           //#sendBuffer.Header.SessionHandle := DWORD_TO_DINT(SWAP(DINT_TO_DWORD(#Config.currentSessionID)));
           #sendBuffer.Header.SessionHandle := DWORD_TO_DINT( SHL(IN := DINT_TO_DWORD(#Config.currentSessionID), N := 24) OR
                                                             (SHL(IN := DINT_TO_DWORD(#Config.currentSessionID), N :=  8) AND DW#16#00FF0000) OR
                                                             (SHR(IN := DINT_TO_DWORD(#Config.currentSessionID), N :=  8) AND DW#16#0000FF00) OR
                                                              SHR(IN := DINT_TO_DWORD(#Config.currentSessionID), N := 24));
           #sendBuffer.Header.Status := 0;
           #sendBuffer.Header.Options := 0;
           //the Context will be a combination out of the own instance identifier
           //and a sequence number
           #sendBuffer.Header.Context[1] := DWORD_TO_BYTE(DINT_TO_DWORD(#ownInstance) AND DW#16#000000FF);
           #sendBuffer.Header.Context[2] := DWORD_TO_BYTE(SHR(IN := DINT_TO_DWORD(#ownInstance), N := 8) AND DW#16#000000FF);
           #sendBuffer.Header.Context[3] := DWORD_TO_BYTE(SHR(IN := DINT_TO_DWORD(#ownInstance), N := 16) AND DW#16#000000FF);
           #sendBuffer.Header.Context[4] := DWORD_TO_BYTE(SHR(IN := DINT_TO_DWORD(#ownInstance), N := 24) AND DW#16#000000FF);
           #sendBuffer.Header.Context[5] := DWORD_TO_BYTE(DINT_TO_DWORD(#ownSequence) AND DW#16#000000FF);
           #sendBuffer.Header.Context[6] := DWORD_TO_BYTE(SHR(IN := DINT_TO_DWORD(#ownSequence), N := 8) AND DW#16#000000FF);
           #sendBuffer.Header.Context[7] := DWORD_TO_BYTE(SHR(IN := DINT_TO_DWORD(#ownSequence), N := 16) AND DW#16#000000FF);
           #sendBuffer.Header.Context[8] := DWORD_TO_BYTE(SHR(IN := DINT_TO_DWORD(#ownSequence), N := 24) AND DW#16#000000FF);
           #sendBuffer.Data[1] := 16#00;

           //Checking the MuteEx
           IF #Config.instanceLock = 0 OR
             #Config.instanceLock = #ownInstance
           THEN
             //Locking the MutEx
             #Config.instanceLock := #ownInstance;
             #send.LEN := #EIP_HEADER_LENGTH;
             #send.REQ := TRUE;
             // Action
             // 

             #send(ID := #connection.id,
                   DATA := #sendBuffer);

             // Transition
             //
             #internalState := #STATE_UNREGISTERING;
             #Config.references := #Config.references - 1;
           ELSE
             IF #Config.instanceLock = #ownInstance THEN
               #Config.instanceLock := 0;
             END_IF;
           END_IF;

         ELSE
           IF #Config.references > 1 THEN
             #Config.references := #Config.references - 1;
           END_IF;
           #internalState := #STATE_POWER_OFF;
         END_IF;

       #STATE_UNREGISTERING:
         // Action
         // 

         #send(ID := #connection.id,
               DATA := #sendBuffer);

         // Transition
         //
         IF #send.STATUS = #RESULT_JOB_START THEN
           ;
         ELSIF #send.STATUS = #RESULT_JOB_RUNNING THEN
           #send.REQ := FALSE;

         ELSIF #send.STATUS = #RESULT_SUCCESS THEN
           #send.REQ := FALSE;
           #internalState := #STATE_DISCONNECTING;
           //Unlocking MuteEx
           #Config.instanceLock := 0;
         ELSE

           #Status := W#16#8200 OR (#send.STATUS AND 16#00FF);
           #send.REQ := FALSE;
           #internalState := #STATE_DISCONNECTING;
         END_IF;

       #STATE_DISCONNECTING:
         IF #disconnect.STATUS = #RESULT_JOB_START THEN
           #connectionStatus.isConnected := FALSE;
           #connectionStatus.isDisconnecting := TRUE;

         ELSIF #disconnect.STATUS = #RESULT_IDLE THEN
           #connectionStatus.isDisconnecting := TRUE;
           #disconnect.REQ := NOT #disconnect.REQ;

         ELSIF #disconnect.STATUS = #RESULT_JOB_RUNNING THEN
           #disconnect.REQ := FALSE;

         ELSIF #disconnect.STATUS = #RESULT_JOB_NOT_REQUIRED OR
           #disconnect.STATUS = #RESULT_SUCCESS
         THEN
           #disconnect.REQ := FALSE;
           #connectionStatus.isConnected := FALSE;
           #connectionStatus.isDisconnecting := FALSE;
           #connectionStatus.isDisconnected := TRUE;
           #connectionStatus.hasReceivedData := FALSE;
           #connectionStatus.hasReceivedHeader := FALSE;

           #ownInstance := 0;
           #ownSequence := 0;
           #Config.connID := 0;

           #internalState := #STATE_IDLE;
         ELSE
           // Throw error !
           //   Error from disconnecting
           #Status := W#16#8400 OR (#disconnect.STATUS AND 16#00FF);
           #disconnect.REQ := FALSE;
           #connectionStatus.isConnected := FALSE;
           #connectionStatus.isDisconnecting := FALSE;
           #connectionStatus.isDisconnected := TRUE;
           #connectionStatus.hasReceivedData := FALSE;
           #connectionStatus.hasReceivedHeader := FALSE;

           #ownInstance := 0;
           #ownSequence := 0;

           #internalState := #STATE_IDLE;
         END_IF;
       ELSE
         // Throw error !
         //   unknown internal state        
         #Status := W#16#8C00 OR (INT_TO_WORD(#internalState) AND W#16#00FF);
     END_CASE;
   END_IF;

   #previousRequest := #REQ;
   #EnabledJ := #Enable;
END_FUNCTION_BLOCK

// folder: GET_PUT_R

FUNCTION_BLOCK "PUT_R"   // FB6, SCL
{ S7_Optimized_Access := 'TRUE' }
VERSION : 1.0
   VAR_INPUT
      Enable : Bool;   // [TRUE| FALSE] TRUE signal keeps the block in PowerOff state
      REQ : Bool;   // [TRUE |FALSE] rising edge triggers a read request
      InterfaceId : Hw_Interface;   // [1..] InterfaceID of the used interface
      IPv4 : IP_V4;   // [IPv4 address] - shall be in the same subnet as controller is
      Slot : Int;   // [-1..16] -1, when directly connected suc has CompactLogix
   END_VAR
   VAR_OUTPUT
      Status : Word;   // [Enum] status information
      Done : Bool;   // [TRUE | FALSE] TRUE signal is a one shot signal indicating the transmission of the data
      Connecting : Bool;   // [TRUE | FALSE] TRUE signal indicates the establishment of the connection
      Established : Bool;   // [TRUE | FALSE] TRUE indicates an established connection
   END_VAR
   VAR_IN_OUT
      Config : "RockwellConfig";
      Tag : "RockwellTag";   // [RockwelTag] datatype containing the tagname, value and data type
      Value : Variant;
   END_VAR
   VAR
      internalState : UInt;   // [Enum] contains the internal state information
      connect : TCON;
      disconnect : TDISCON;
      send : TSEND;
      receive : TRCV;
      diag : T_DIAG;
      connection : TCON_IP_v4;
      sendBuffer : Struct
         Header : Struct
            Command : Word;   // Encapsulation command
            Length : UInt;   // Length, in bytes, of the command specific data portion of the message
            SessionHandle : UDInt;   // Session identification
            Status : UDInt;   // Status code
            Context : Array[1..8] of USInt;   // Information pertinien only to the sender of an encapsulation command
            Options : UDInt;
         END_STRUCT;
         Data : Array[1..508] of USInt;
      END_STRUCT;
      receiveBuffer : Struct
         Header : Struct
            Command : Word;   // Encapsulation command
            Length : UInt;   // Length, in bytes, of the command specific data portion of the message
            SessionHandle : UDInt;   // Session identification
            Status : UDInt;   // Status code
            Context : Array[1..8] of USInt;   // Information pertinien only to the sender of an encapsulation command
            Options : UDInt;
         END_STRUCT;
         Data : Array[1..508] of USInt;
      END_STRUCT;
      currentResponse : Word;
      connectionStatus : Struct
         isDisconnected : Bool;
         isDisconnecting : Bool;
         isConnecting : Bool;
         isConnected : Bool;
         hasReceivedData : Bool;
         hasReceivedHeader : Bool;
      END_STRUCT;
      indexTag : Int := 0;
      currentCIPService : Byte;
      previousRequest : Bool;
      EnabledJ : Bool;
      ownInstance : DInt;
      ownSequence : DInt;
      diagStatus : TDiag_StatusExt;
      randomGenerator : Struct   // [STRUCT] used to realize a pseudo random number
         m_w : DInt;
         m_z : DInt;
         Val : DInt;
         currentTime : DTL;
         currentMilliSeconds : DInt;
      END_STRUCT;
   END_VAR
   VAR_TEMP
      indexTagName : DInt;
      result : Int;
      itemLength : DInt;   // contains the Length of the EIP packet
      overallLength : DInt;   // contains the Length of the EIP packet
      tagNameLength : DInt;   // contains the Length of the Tagname (in WORDS)
      tagValueLength : DInt;   // contains the Length of the Tag Value
      unconnectedDataItemLength : DInt;   // contains the Length of the unconnected data item
      baseIndexOuterCIPMessage : DInt;   // contains the base index to the beginning of the outer CIP message
      baseIndexInnerCIPMessage : DInt;   // contains the base index to the beginning of the inner CIP message
      receivedServiceStatus : Int;
      receivedInstance : DInt;
      receivedSequence : DInt;
      receivedType : Word;
      valueIndex : Int;
      sendValue : Struct
         Boolean : Bool;
         Short : SInt;
         Integer : Int;
         Double : DInt;
         Float : Real;
      END_STRUCT;
   END_VAR
   VAR CONSTANT
      EIP_VENDOR_ID : Word := 1251;   // EtherNet/IP vendor ID 'Siemens AG'
      EIP_HEADER_LENGTH : UInt := 24;   // EtherNet/IP Encapsulation Header length is 24 bytes
      EIP_PORT : Word := 44818;   // EtherNet/IP standard port is 44818 (0xAF12)
      RESULT_SUCCESS : Word := 16#0000;
      RESULT_IDLE : Word := 16#7000;
      RESULT_JOB_START : Word := 16#7001;
      RESULT_JOB_RUNNING : Word := 16#7002;
      RESULT_JOB_NOT_REQUIRED : Word := 16#80A3;
      RESULT_MORE_AVAIL : Word := 16#80B1;
      RESULT_REUSED_ID : Word := 16#8085;
      EIP_STATUS_OK : UDInt := 0;   // EIP Status OK
      EIP_STATUS_TOOMANY_SESSIONS : UDInt := 16#01000000;   // EIP Status "more than 1 active session on the same TCP connection"
      EIP_STATUS_OUTOFRESSOURCES : UDInt := 16#02000000;   // EIP Status "does not have sufficient resources"
      EIP_STATUS_INVALID_SESSION_ID : UDInt := 16#64000000;   // EIP Status "Invalid Session ID"
      EIP_STATUS_PROTOCOL_ERROR : UDInt := 16#69000000;   // EIP Status "Protocol Version or Options mismatches"
      EIP_CMD_REG_SESSION : Word := 16#0065;   // EtherNet/IP Encapsulation Command "Register Session"
      EIP_CMD_UNREG_SESSION : Word := 16#0066;   // EtherNet/IP Encapsulation Command "Unregister Session"
      EIP_CMD_SEND_RR : Word := 16#006F;   // EtherNet/IP Encapsulation Command "Send RR Data"
      CIP_SRV_TABLEREAD : Byte := 16#4C;   // CIP Service Data Table Read
      CIP_SRV_TABLEWRITE : Byte := 16#4D;   // CIP Service Data Table Write
      CIP_SRV_TABLEREAD_FRAG : Byte := 16#52;   // CIP Service Fragmented Data Table Read
      CIP_SRV_TABLEWRITE_FRAG : Byte := 16#53;   // CIP Service Fragmented Data Table Write
      CIP_SRV_UNCONNECTED_SEND : Byte := 16#52;   // CIP Service Unconnected Send Data
      STATE_IDLE : UInt := 1;
      STATE_INIT : UInt := 2;
      STATE_CONNECTING : UInt := 3;
      STATE_DISCONNECTING : UInt := 4;
      STATE_SENDING : UInt := 5;
      STATE_REGISTER_SESSION : UInt := 6;
      STATE_UNREGISTER_SESSION : UInt := 7;
      STATE_REGISTERING : UInt := 8;
      STATE_UNREGISTERING : UInt := 9;
      STATE_REGISTERED : UInt := 10;
      STATE_SEND : UInt := 11;
      STATE_RECEIVE_HEADER : UInt := 12;
      STATE_RECEIVE_DATA : UInt := 13;
      STATE_POWER_OFF : UInt := 0;
      DT_BOOLEAN_ATOMIC : USInt := 16#C1;
      DT_SINT_ATOMIC : USInt := 16#C2;
      DT_INT_ATOMIC : USInt := 16#C3;
      DT_DINT_ATOMIC : USInt := 16#C4;
      DT_FLOAT_ATOMIC : USInt := 16#CA;
      CIP_PATH_SEG_TYPE_CLASS : USInt := 16#20;
      CIP_PATH_SEG_TYPE_INSTANCE : USInt := 16#24;
      CIP_PATH_SEG_TYPE_ANSI : USInt := 16#91;
      CIP_PATH_SEG_TYPE_PORT : USInt := 16#01;
      CIP_ROUTE_SEG_LENGTH : Int := 4;
      CIP_ROUTE_PATH_LENGTH : Int := 1;
      CIP_TABLEREAD_LENGTH : Int := 6;
      CIP_TABLEWRITE_LENGTH : Int := 4;
      CIP_UCSEND_HEADER_LENGTH : Int := 4;
      CIP_UCSEND_SEG_LENGTH : Int := 6;
      EIP_CMD_SEND_RR_SEG_LENGTH : Int := 16;
      CON_TYPE_TCP_V2 : USInt := 17;   // TCP connection for TCON_PARAM descriptor
      CON_TYPE_TCP_V4 : Byte := 11;   // TCP connection for TCON_IP_V4 descriptor
      CIP_GENSTS_SUCCESS : USInt := 16#00;
      CIP_GENSTS_PATH_SEG_ERROR : USInt := 16#04;
      CIP_GENSTS_PATH_DEST_UNKNOWN : USInt := 16#05;
      CIP_GENSTS_PARTIAL : USInt := 16#06;
      CIP_GENSTS_NOT_ENOUGH_DATA : USInt := 16#13;
      CIP_GENSTS_PATH_SIZE_MISMATCH : USInt := 16#26;
      CIP_GENSTS_DOESNT_EXIST : USInt := 16#16;
      CIP_GENSTS_GENERIC : USInt := 16#FF;
      CIP_SRVSTS_RANGE_EXCEED : UInt := 16#2105;
      CIP_SRVSTS_TYPE_MISMATCH : UInt := 16#2107;
   END_VAR
BEGIN
   //=============================================================================
   // Siemens AG
   // (c)Copyright 2016 All Rights Reserved
   //-----------------------------------------------------------------------------
   // Library: PutGet_Rockwell
   // Tested with: 1511-1 PN V1.8.3 and ControlLogix/Compactlogix
   // Engineering: TIA Portal V13 SP1 Upd 9
   // Restrictions: look into pdf
   // Requirements: S7-1500 V1.8.3
   // Functionality: Get Put Values from to Rockwell CPU
   //-----------------------------------------------------------------------------
   // Change log table:
   // Version  Date            Expert in charge        Changes applied
   // 01.00.01 12.07.2016      Scheel                  initial version 
   // 01.00.02 22.07.2016      Scheel                  feat: add diagnostics and
   //                                                        indicators
   // 01.00.03 22.07.2016      Scheel                  fix: diagnostics indicators
   // 01.00.04 19.10.2016      Scheel                  fix: connect will be
   //                                                       retriggered, when idle
   //                                                  refac: change of IP address
   //                                                         datatype to IP_V4
   //                                                  feat: add recognition of
   //                                                        CIP specific status
   //=============================================================================
   //

   //#########################################################################################
   // Pseudo Random number generator
   //
   //  This Random number function generator is based on multiplication and
   //  addition with overflow invented by George Marsaglia.
   //  The loss of information is intended.
   //  
   //  Wikipedia (https://en.wikipedia.org/wiki/Random_number_generation)
   //#########################################################################################
   //
   //Initialization of the variables using a time value as a seed
   #result := RD_SYS_T(#randomGenerator.currentTime);
   #randomGenerator.currentMilliSeconds := UDINT_TO_DINT(#randomGenerator.currentTime.NANOSECOND) / 1000000 + (USINT_TO_DINT(#randomGenerator.currentTime.SECOND) * 1000);

   IF #randomGenerator.m_w = 0 OR #randomGenerator.m_z = 0 THEN
     #randomGenerator.m_w := UDINT_TO_DINT((#randomGenerator.currentTime.NANOSECOND / 1000000)) + 2;    // using the milliseconds since the PLC has been powered on
     #randomGenerator.m_z := 13696;
   ELSE
     #randomGenerator.m_z := 36969 * DWORD_TO_DINT(DINT_TO_DWORD(#randomGenerator.m_z) AND 16#FFFF)
     + DWORD_TO_DINT(SHR(IN := DINT_TO_DWORD(#randomGenerator.m_z), N := 16));
     #randomGenerator.m_w := 18000 * DWORD_TO_DINT(DINT_TO_DWORD(#randomGenerator.m_w) AND 16#FFFF)
     + DWORD_TO_DINT(SHR(IN := DINT_TO_DWORD(#randomGenerator.m_w), N := 16));
     #randomGenerator.Val := DWORD_TO_DINT(SHL(IN := DINT_TO_DWORD(#randomGenerator.m_z), N := 16)) + #randomGenerator.m_w;  // 32-bit result */    
   END_IF;

   //assume sane state
   #Status := #RESULT_IDLE;
   #Done := FALSE;

   #connect(ID := #connection.ID,
            CONNECT := #connection);

   #disconnect(ID := #connection.ID);


   IF NOT #Enable AND #EnabledJ THEN
     // Complete Restart detected 
     //
     #internalState := #STATE_UNREGISTER_SESSION;

   ELSIF #Enable AND NOT #EnabledJ THEN
     #internalState := #STATE_INIT;

   ELSE
     // Regular operation
     //   
     CASE #internalState OF
       #STATE_POWER_OFF:
         //Preset the TCP connection information
         //  
         IF #Config.connID = 0 THEN
           #Config.connID := DWORD_TO_WORD(DINT_TO_DWORD((#randomGenerator.Val MOD 2048) + 2048));
         END_IF;
         #connection.ID := #Config.connID;

         // only usable in S7-1500 or S7-1200 V4.x
         // 
         #connection.ConnectionType := #CON_TYPE_TCP_V4;           //TCP connection
         #connection.InterfaceId := #InterfaceId;
         #connection.ActiveEstablished := TRUE;             //active connection (Client)

         #connection.RemoteAddress := #IPv4;

         #connection.RemotePort := WORD_TO_UINT(#EIP_PORT);

         // #connection.CONNECTION_TYPE := #CON_TYPE_TCP_V2;      //TCP connection
         // #connection.LOCAL_DEVICE_ID := WORD_TO_USINT(#InterfaceId);
         // #connection.ACTIVE_EST := TRUE;                //active connection (Client)

         // #connection.REM_STADDR_LEN := 4;
         // #connection.REM_STADDR[1] := BYTE_TO_USINT(#IPv4[1]);
         // #connection.REM_STADDR[2] := BYTE_TO_USINT(#IPv4[2]);
         // #connection.REM_STADDR[3] := BYTE_TO_USINT(#IPv4[3]);
         // #connection.REM_STADDR[4] := BYTE_TO_USINT(#IPv4[4]);

         // #connection.REM_TSAP_ID_LEN := 2;
         // #connection.REM_TSAP_ID[1] := WORD_TO_BYTE(SHR(IN := #EIP_PORT, N := 8));
         // #connection.REM_TSAP_ID[2] := WORD_TO_BYTE(#EIP_PORT AND W#16#FF);

         #ownInstance := 0;
         #ownSequence := 0;

         #internalState := #STATE_IDLE;

       #STATE_IDLE:

         // Action
         // 
         #Done := FALSE;

         // Transition 
         //IF NOT #connectionStatus.isConnected THEN
         //  #internalState := #STATE_INIT;          
         IF #connectionStatus.isConnected AND #REQ AND NOT #previousRequest AND #Enable THEN
           #internalState := #STATE_SENDING;
           #Status := #RESULT_JOB_START;
         END_IF;


       #STATE_INIT:
         //Preset the TCP connection information
         //
         IF #Config.connID = 0 THEN
           #Config.connID := DWORD_TO_WORD(DINT_TO_DWORD((#randomGenerator.Val MOD 2048) + 2048));
         END_IF;
         #connection.ID := #Config.connID;

         //Inserting Semaphore checking
         //
         //  Only issue a new connect, when there is no one is referencing the connection already
         //  Otherwise just skip that step and use the established connection
         //  

         IF #Config.references = 0 THEN
           // only usable in S7-1500 or S7-1200 V4.x
           // 
           #connection.ConnectionType := #CON_TYPE_TCP_V4;    //TCP connection
           #connection.InterfaceId := #InterfaceId;
           #connection.ActiveEstablished := TRUE;             //active connection (Client)

           #connection.RemoteAddress := #IPv4;

           #connection.RemotePort := WORD_TO_UINT(#EIP_PORT);

           // #connection.CONNECTION_TYPE := #CON_TYPE_TCP_V2;      //TCP connection
           // #connection.LOCAL_DEVICE_ID := WORD_TO_USINT(#InterfaceId);
           // #connection.ACTIVE_EST := TRUE;                //active connection (Client)

           // #connection.REM_STADDR_LEN := 4;
           // #connection.REM_STADDR[1] := BYTE_TO_USINT(#IPv4[1]);
           // #connection.REM_STADDR[2] := BYTE_TO_USINT(#IPv4[2]);
           // #connection.REM_STADDR[3] := BYTE_TO_USINT(#IPv4[3]);
           // #connection.REM_STADDR[4] := BYTE_TO_USINT(#IPv4[4]);

           // #connection.REM_TSAP_ID_LEN := 2;
           // #connection.REM_TSAP_ID[1] := WORD_TO_BYTE(SHR(IN := #EIP_PORT, N := 8));
           // #connection.REM_TSAP_ID[2] := WORD_TO_BYTE(#EIP_PORT AND W#16#FF);


           //No connection established yet
           //  issue a new request
           #connect.REQ := TRUE;
           #internalState := #STATE_CONNECTING;
         ELSE
           #internalState := #STATE_IDLE;
           #connectionStatus.isConnected := TRUE;
         END_IF;
         #Config.references := #Config.references + 1;

         //Remember the currently active instance reference as my own instance identifier
         //  and reset the Sequence counter
         #ownInstance := #Config.references;
         #ownSequence := 0;

       #STATE_CONNECTING:

         IF #connect.STATUS = #RESULT_JOB_START THEN
           #connectionStatus.isConnecting := TRUE;
         ELSIF #connect.STATUS = #RESULT_IDLE THEN
           #connect.REQ := NOT #connect.REQ;

         ELSIF #connect.STATUS = #RESULT_JOB_RUNNING THEN
           #connect.REQ := FALSE;

         ELSIF #connect.STATUS = #RESULT_JOB_NOT_REQUIRED OR
               #connect.STATUS = #RESULT_SUCCESS 
         THEN
           #connect.REQ := FALSE;
           #connectionStatus.isConnecting := FALSE;
           #connectionStatus.isConnected := TRUE;
           #connectionStatus.isDisconnected := FALSE;

           #internalState := #STATE_REGISTER_SESSION;

         ELSE
           // Throw error !
           //   Error in connect
           #Status := W#16#8100 OR (#connect.STATUS AND 16#00FF);   //Error in connecting       
           #connect.REQ := FALSE;
           #internalState := #STATE_DISCONNECTING;
         END_IF;

       #STATE_REGISTER_SESSION:

         #sendBuffer.Header.Command := SWAP(#EIP_CMD_REG_SESSION);                                                 //Command is RegisterSession (16#65)
         #sendBuffer.Header.Length  := WORD_TO_UINT(SWAP(IN := UDINT_TO_WORD(4)));    //Length of Data is 4 Bytes
         #sendBuffer.Header.SessionHandle := 0;
         #sendBuffer.Header.Status := 0;
         #sendBuffer.Header.Options := 0;
         //the Context will be a combination out of the own instance identifier
         //and a sequence number
         #sendBuffer.Header.Context[1] := DWORD_TO_USINT(DINT_TO_DWORD(#ownInstance) AND DW#16#000000FF);
         #sendBuffer.Header.Context[2] := DWORD_TO_USINT(SHR(IN := DINT_TO_DWORD(#ownInstance), N := 8) AND DW#16#000000FF);
         #sendBuffer.Header.Context[3] := DWORD_TO_USINT(SHR(IN := DINT_TO_DWORD(#ownInstance), N := 16) AND DW#16#000000FF);
         #sendBuffer.Header.Context[4] := DWORD_TO_USINT(SHR(IN := DINT_TO_DWORD(#ownInstance), N := 24) AND DW#16#000000FF);
         #sendBuffer.Header.Context[5] := DWORD_TO_USINT(DINT_TO_DWORD(#ownSequence) AND DW#16#000000FF);
         #sendBuffer.Header.Context[6] := DWORD_TO_USINT(SHR(IN := DINT_TO_DWORD(#ownSequence), N := 8) AND DW#16#000000FF);
         #sendBuffer.Header.Context[7] := DWORD_TO_USINT(SHR(IN := DINT_TO_DWORD(#ownSequence), N := 16) AND DW#16#000000FF);
         #sendBuffer.Header.Context[8] := DWORD_TO_USINT(SHR(IN := DINT_TO_DWORD(#ownSequence), N := 24) AND DW#16#000000FF);
         #sendBuffer.Data[1] := 16#01;                                 //Protocol Version V1.0

         //Checking the MuteEx
         IF #Config.instanceLock = 0 OR
           #Config.instanceLock = #ownInstance
         THEN
           //allowed to utilize, since instanceLock is either 0 or ownInstance
           #send(ID := #connection.ID,
                 DATA := #sendBuffer);

           //Locking the MutEx
           #Config.instanceLock := #ownInstance;
           #send.LEN := #EIP_HEADER_LENGTH + 4;
           #send.REQ := TRUE;

           #internalState := #STATE_REGISTERING;
         ELSE
           ;
         END_IF;

       #STATE_REGISTERING:
         // Action
         // 

         //allowed to utilize, since instanceLock is either 0 or ownInstance
         #send(ID := #connection.ID,
               DATA := #sendBuffer);

         // Transition
         // 
         IF #send.STATUS = #RESULT_JOB_START THEN
           ;
         ELSIF #send.STATUS = #RESULT_JOB_RUNNING THEN
           #send.REQ := FALSE;

         ELSIF #send.STATUS = #RESULT_IDLE THEN
           #send.REQ := NOT #send.REQ;

         ELSIF #send.STATUS = #RESULT_SUCCESS THEN
           #send.REQ := FALSE;
           #internalState := #STATE_RECEIVE_HEADER;
         ELSE
           // Throw error !
           //   in Registering
           #Status := W#16#8200 OR (#send.STATUS AND 16#00FF);   //Error in sending
           #send.REQ := FALSE;
           #internalState := #STATE_DISCONNECTING;
         END_IF;

       #STATE_SENDING:
         #sendBuffer.Header.Command := SWAP(#EIP_CMD_SEND_RR);                                                 //Command is SendRRData (16#6F)
         //
         // overall Message length depends on the packet content and is therefore assigned later
         //
         #sendBuffer.Header.SessionHandle := DWORD_TO_UDINT(SWAP(UDINT_TO_DWORD(#Config.currentSessionID)));;
         #sendBuffer.Header.Status := 0;
         #sendBuffer.Header.Options := 0;
         //the Context will be a combination out of the own instance identifier
         //and a sequence number
         #sendBuffer.Header.Context[1] := DWORD_TO_USINT(DINT_TO_DWORD(#ownInstance) AND DW#16#000000FF);
         #sendBuffer.Header.Context[2] := DWORD_TO_USINT(SHR(IN := DINT_TO_DWORD(#ownInstance), N := 8) AND DW#16#000000FF);
         #sendBuffer.Header.Context[3] := DWORD_TO_USINT(SHR(IN := DINT_TO_DWORD(#ownInstance), N := 16) AND DW#16#000000FF);
         #sendBuffer.Header.Context[4] := DWORD_TO_USINT(SHR(IN := DINT_TO_DWORD(#ownInstance), N := 24) AND DW#16#000000FF);
         #sendBuffer.Header.Context[5] := DWORD_TO_USINT(DINT_TO_DWORD(#ownSequence) AND DW#16#000000FF);
         #sendBuffer.Header.Context[6] := DWORD_TO_USINT(SHR(IN := DINT_TO_DWORD(#ownSequence), N := 8) AND DW#16#000000FF);
         #sendBuffer.Header.Context[7] := DWORD_TO_USINT(SHR(IN := DINT_TO_DWORD(#ownSequence), N := 16) AND DW#16#000000FF);
         #sendBuffer.Header.Context[8] := DWORD_TO_USINT(SHR(IN := DINT_TO_DWORD(#ownSequence), N := 24) AND DW#16#000000FF);
         //CIP specific data
         #sendBuffer.Data[1] := 16#0;                                 //CIP Interface handle
         #sendBuffer.Data[2] := 16#0;
         #sendBuffer.Data[3] := 16#0;
         #sendBuffer.Data[4] := 16#0;

         #sendBuffer.Data[5] := 16#0;                                  //Timeout
         #sendBuffer.Data[6] := 16#0;

         #sendBuffer.Data[7] := 16#2;                                  //Items
         #sendBuffer.Data[8] := 16#0;

         #sendBuffer.Data[9] := 16#0;                                  //Null address item
         #sendBuffer.Data[10] := 16#0;
         #sendBuffer.Data[11] := 16#0;                                  //Null address item Length = 0
         #sendBuffer.Data[12] := 16#0;

         #sendBuffer.Data[13] := 16#B2;                                  //Unconnected data item
         #sendBuffer.Data[14] := 16#0;
         //Item Length needs to be added, but since that depends on the content,
         //it will will be assigned later. It occupies 2 Bytes, thus the outer CIP Message 
         //starts at offset 17 into the Data (1 based counting)
         //
         #baseIndexOuterCIPMessage := 17;

         //CIP Message
         //  here a decision needs to be made
         //  In case Slot is -1 a direct connection is assumed, such as for a CompactLogix, this means no
         //  further route segments are necessary
         //  In case Slot is anywhere between 0 and 16 a route segment is required, since the CPU is not
         //  identical to the ethernet interface, as in a ControlLogix L5, L6, L7 series system

         //Length of the following Path segment depends only on the length of the Tagname measured in WORDS
         // plus 1 WORD for the segment encoding information
         // 
         #tagNameLength := ((LEN(#Tag."Name") + 1) / 2) * 2;

         //
         //  Prelude
         //
         //In case the slot information is negative (-1) there is no additional path segment
         //Any other slot value requires routing information, which need to be added
         //  this means the preparation of offsets and header needs to be done, before
         //  the common part of copying the value to the packet can take place
         IF #Slot = -1 THEN
           //directly connected (onboard) Ethernet interface
           //
           #baseIndexInnerCIPMessage := #baseIndexOuterCIPMessage;

         ELSE
           //not directly connected (through external) Ethernet interface
           //
           //  preparing offsets for length calculation as well as header
           //  There is a 10 byte segment before the tag value segment
           #baseIndexInnerCIPMessage := #baseIndexOuterCIPMessage + 10;

           #sendBuffer.Data[#baseIndexOuterCIPMessage]     := BYTE_TO_USINT(#CIP_SRV_UNCONNECTED_SEND);  //CIP service = UNCONNECTED_SEND_DATA = 16#52
           #sendBuffer.Data[#baseIndexOuterCIPMessage + 1] := 2;                                     //Path Size is constant 2 WORDS

           #sendBuffer.Data[#baseIndexOuterCIPMessage + 2] := #CIP_PATH_SEG_TYPE_CLASS;              //Path Type = Class Segment
           #sendBuffer.Data[#baseIndexOuterCIPMessage + 3] := 16#06;                                 //Class = ConnectionManager (16#06)

           #sendBuffer.Data[#baseIndexOuterCIPMessage + 4] := #CIP_PATH_SEG_TYPE_INSTANCE;           //Path Type = Instance Segment
           #sendBuffer.Data[#baseIndexOuterCIPMessage + 5] := 16#01;                                 //Instance =Instance 1 (16#01)

           //Encapsulated CIP Message
           //
           #sendBuffer.Data[#baseIndexOuterCIPMessage + 6] := 16#07;                                 //Priority combined with TimeTick (= 16#07)
           #sendBuffer.Data[#baseIndexOuterCIPMessage + 7] := INT_TO_USINT(233);                     //???

         END_IF;

         //
         // tag value segment
         // 

         #sendBuffer.Data[#baseIndexInnerCIPMessage]     := BYTE_TO_USINT(#CIP_SRV_TABLEWRITE);     //CIP service = DATA_TABLE_READ = 16#4D

         #sendBuffer.Data[#baseIndexInnerCIPMessage + 1] := DINT_TO_USINT(#tagNameLength / 2 + 1);  //Path Size
         #sendBuffer.Data[#baseIndexInnerCIPMessage + 2] := #CIP_PATH_SEG_TYPE_ANSI;                //Path Type = ANSI Extended Symbol Segment

         //Copy In
         #sendBuffer.Data[#baseIndexInnerCIPMessage + 3] := INT_TO_USINT(LEN(#Tag."Name"));          //TagName Length (bytes)
         FOR #indexTagName := 1 TO USINT_TO_INT(#sendBuffer.Data[#baseIndexInnerCIPMessage + 3]) DO
           #sendBuffer.Data[#baseIndexInnerCIPMessage + 3 + #indexTagName] := CHAR_TO_USINT(#Tag."Name"[#indexTagName]);
         END_FOR;

         //in case the tag name has an odd (uneven) length the path segment content needs to be padded to be WORD aligned
         //
         #indexTagName := #indexTagName - 1;
         IF #indexTagName MOD 2 <> 0 THEN
           #indexTagName := #indexTagName + 1;
           #sendBuffer.Data[#baseIndexInnerCIPMessage + 3 + #indexTagName] := 0;
         END_IF;

         //Command Specific information
         //
         #sendBuffer.Data[#baseIndexInnerCIPMessage + 4 + #indexTagName] := INT_TO_USINT(#Tag.DataType);
         #sendBuffer.Data[#baseIndexInnerCIPMessage + 5 + #indexTagName] := 0;
         #sendBuffer.Data[#baseIndexInnerCIPMessage + 6 + #indexTagName] := INT_TO_USINT(#Tag.Count);                 //number of values to follow
         #sendBuffer.Data[#baseIndexInnerCIPMessage + 7 + #indexTagName] := WORD_TO_USINT(SHR(IN := INT_TO_WORD(#Tag.Count), N := 8) AND W#16#00FF);

         //for testing purposes only
         #valueIndex := 0;

         WHILE #valueIndex <= #Tag.Count DO

           //Copy the value in, type dependant
           IF #Tag.DataType = #DT_BOOLEAN_ATOMIC THEN
             //Transferring the Value
             //
             // There seems to be a difficultiy with accessing boolean variables, the 
             // access need to be provided as accesses to byte (SINT)
             // 16#FF == TRUE
             // 16#00 == FALSE
             // 
             #result := MOVE_BLK_VARIANT(COUNT := 1,
                                         SRC := #Value,
                                         SRC_INDEX := #valueIndex,
                                         DEST_INDEX := 0,
                                         DEST => #sendValue.Short);
             #sendBuffer.Data[#baseIndexInnerCIPMessage + 8 + #indexTagName + #valueIndex] := SINT_TO_USINT(#sendValue.Short);
             #tagValueLength := (4 + ((#Tag.Count + 1) / 2) * 2) * 1;

           ELSIF #Tag.DataType = #DT_SINT_ATOMIC THEN
             //Transferring the Value
             //
             #result := MOVE_BLK_VARIANT(COUNT := 1,
                                         SRC := #Value,
                                         SRC_INDEX := #valueIndex,
                                         DEST_INDEX := 0,
                                         DEST => #sendValue.Short);
             #sendBuffer.Data[#baseIndexInnerCIPMessage + 8 + #indexTagName + #valueIndex] := SINT_TO_USINT(#sendValue.Short);
             #tagValueLength := (4 + ((#Tag.Count + 1)/ 2) * 2) * 1;

           ELSIF #Tag.DataType = #DT_INT_ATOMIC THEN
             //Transferring the Value
             //
             #result := MOVE_BLK_VARIANT(COUNT := 1,
                                         SRC := #Value,
                                         SRC_INDEX := #valueIndex,
                                         DEST_INDEX := 0,
                                         DEST => #sendValue.Integer);
             #sendBuffer.Data[#baseIndexInnerCIPMessage + 8 + #indexTagName + #valueIndex * 2] := BYTE_TO_USINT(DWORD_TO_BYTE(          INT_TO_WORD(#sendValue.Integer) AND B#16#FF));
             #sendBuffer.Data[#baseIndexInnerCIPMessage + 9 + #indexTagName + #valueIndex * 2] := BYTE_TO_USINT(DWORD_TO_BYTE(SHR(IN := INT_TO_WORD(#sendValue.Integer), N := 8)));

             #tagValueLength := 4 + #Tag.Count * 2;
           ELSIF #Tag.DataType = #DT_DINT_ATOMIC THEN
             //Transferring the Value
             //
             #result := MOVE_BLK_VARIANT(COUNT := 1,
                                         SRC := #Value,
                                         SRC_INDEX := #valueIndex,
                                         DEST_INDEX := 0,
                                         DEST => #sendValue.Double);
             #sendBuffer.Data[#baseIndexInnerCIPMessage +  8 + #indexTagName + #valueIndex * 4] := BYTE_TO_USINT(DWORD_TO_BYTE(          DINT_TO_DWORD(#sendValue.Double) AND B#16#FF));
             #sendBuffer.Data[#baseIndexInnerCIPMessage +  9 + #indexTagName + #valueIndex * 4] := BYTE_TO_USINT(DWORD_TO_BYTE(SHR(IN := DINT_TO_DWORD(#sendValue.Double), N := 8)));
             #sendBuffer.Data[#baseIndexInnerCIPMessage + 10 + #indexTagName + #valueIndex * 4] := BYTE_TO_USINT(DWORD_TO_BYTE(SHR(IN := DINT_TO_DWORD(#sendValue.Double), N := 16)));
             #sendBuffer.Data[#baseIndexInnerCIPMessage + 11 + #indexTagName + #valueIndex * 4] := BYTE_TO_USINT(DWORD_TO_BYTE(SHR(IN := DINT_TO_DWORD(#sendValue.Double), N := 24)));

             #tagValueLength := 4 + #Tag.Count * 4;

           ELSIF #Tag.DataType = #DT_FLOAT_ATOMIC THEN
               //Transferring the Value
               //
               #result := MOVE_BLK_VARIANT(COUNT := 1,
                                           SRC := #Value,
                                           SRC_INDEX := #valueIndex,
                                           DEST_INDEX := 0,
                                           DEST => #sendValue.Float);
               #sendBuffer.Data[#baseIndexInnerCIPMessage +  8 + #indexTagName + #valueIndex * 4] := BYTE_TO_USINT(DWORD_TO_BYTE(          REAL_TO_DWORD(#sendValue.Float) AND B#16#FF));
               #sendBuffer.Data[#baseIndexInnerCIPMessage +  9 + #indexTagName + #valueIndex * 4] := BYTE_TO_USINT(DWORD_TO_BYTE(SHR(IN := REAL_TO_DWORD(#sendValue.Float), N := 8)));
               #sendBuffer.Data[#baseIndexInnerCIPMessage + 10 + #indexTagName + #valueIndex * 4] := BYTE_TO_USINT(DWORD_TO_BYTE(SHR(IN := REAL_TO_DWORD(#sendValue.Float), N := 16)));
               #sendBuffer.Data[#baseIndexInnerCIPMessage + 11 + #indexTagName + #valueIndex * 4] := BYTE_TO_USINT(DWORD_TO_BYTE(SHR(IN := REAL_TO_DWORD(#sendValue.Float), N := 24)));
           ELSE
             //Throw error
             //  - unknown/ unsupported data type specified
             //  
             // throw warning
             #Status := 16#7303; //Unknown data type
             #tagValueLength := 0;
           END_IF;
           #valueIndex := #valueIndex + 1;
         END_WHILE;

         #itemLength := #tagNameLength + #tagValueLength + + #CIP_TABLEWRITE_LENGTH;

         //
         // Closure
         //

         IF #Slot = -1 THEN
           #unconnectedDataItemLength := #itemLength;
         ELSE
           #sendBuffer.Data[#baseIndexOuterCIPMessage + 8] := WORD_TO_USINT(DINT_TO_WORD(#itemLength));                  //Unconnected data item Length
           #sendBuffer.Data[#baseIndexOuterCIPMessage + 9] := WORD_TO_USINT(SHL(IN := DINT_TO_WORD(#itemLength), N := 8));  //Unconnected data item Length

           //Routing Information
           #sendBuffer.Data[#baseIndexInnerCIPMessage + #itemLength] := INT_TO_USINT(#CIP_ROUTE_PATH_LENGTH);
           #sendBuffer.Data[#baseIndexInnerCIPMessage + #itemLength + 1] := 0;

           #sendBuffer.Data[#baseIndexInnerCIPMessage + #itemLength + 2] := #CIP_PATH_SEG_TYPE_PORT;
           #sendBuffer.Data[#baseIndexInnerCIPMessage + #itemLength + 3] := INT_TO_USINT(#Slot);



           #unconnectedDataItemLength := #itemLength
                                       + #CIP_ROUTE_SEG_LENGTH
                                       + #CIP_UCSEND_HEADER_LENGTH
                                       + #CIP_UCSEND_SEG_LENGTH;
         END_IF;

         //Length of the unconnected data item depends on the content of the package
         //
         #sendBuffer.Data[15] := WORD_TO_USINT(        DINT_TO_WORD(#unconnectedDataItemLength));        //Unconnected data item Length
         #sendBuffer.Data[16] := WORD_TO_USINT(SHL(IN:=DINT_TO_WORD(#unconnectedDataItemLength),N:=8));  //Unconnected data item Length

         #sendBuffer.Header.Length := WORD_TO_UINT(SWAP(IN := DINT_TO_WORD(#unconnectedDataItemLength + #EIP_CMD_SEND_RR_SEG_LENGTH)));    //Length of Data

         //Checking the MuteEx
         IF #Config.instanceLock = 0 OR
           #Config.instanceLock = #ownInstance
         THEN
           #Config.instanceLock := #ownInstance;
           #send.LEN := DINT_TO_UINT(#EIP_HEADER_LENGTH + #unconnectedDataItemLength + #EIP_CMD_SEND_RR_SEG_LENGTH);
           #send.REQ := TRUE;

           //allowed to utilize, since instanceLock is either 0 or ownInstance
           #send(ID := #connection.ID,
                 DATA := #sendBuffer);

           #internalState := #STATE_SEND;
         ELSE
           ;
         END_IF;
         #Status := #RESULT_JOB_RUNNING;

       #STATE_SEND:
         // Action
         //

         // assume job is still running
         #Status := #RESULT_JOB_RUNNING;

         #send(ID := #connection.ID,
               DATA := #sendBuffer);

         // Transition
         //
         IF #send.STATUS = #RESULT_JOB_START THEN
           ;

         ELSIF #send.STATUS = #RESULT_IDLE THEN
           #send.REQ := NOT #send.REQ;

         ELSIF #send.STATUS = #RESULT_JOB_RUNNING THEN
           #send.REQ := FALSE;

         ELSIF #send.STATUS = #RESULT_SUCCESS THEN
           #send.REQ := FALSE;
           #internalState := #STATE_RECEIVE_HEADER;

         ELSE
           // Throw error !
           // 
           #Status := W#16#8200 OR (#send.STATUS AND 16#00FF);
           #send.REQ := FALSE;
           #internalState := #STATE_DISCONNECTING;
         END_IF;

       #STATE_RECEIVE_HEADER:
         // Action
         // Receive Header data
         // 

         // assume job is still running
         #Status := #RESULT_JOB_RUNNING;

         #receive(EN_R := (#ownInstance = #Config.instanceLock),
                  ID := #connection.ID,
                  LEN := #EIP_HEADER_LENGTH,
                  DATA := #receiveBuffer.Header);


         // Transition
         // Header received --> STATE_RECEIVE_DATA
         // Invalid Data --> IDLE
         // Error --> INIT
         IF #receive.NDR OR #receive.STATUS = #RESULT_SUCCESS THEN
           IF #receiveBuffer.Header.Length = 0 THEN
             //Unlocking MuteEx
             #Config.instanceLock := 0;
             #internalState := #STATE_IDLE;
           ELSE
             #internalState := #STATE_RECEIVE_DATA;
           END_IF;
         ELSIF #receive.STATUS <> #RESULT_IDLE AND
           #receive.STATUS <> #RESULT_JOB_RUNNING AND
           #receive.STATUS <> #RESULT_JOB_START AND
           #receive.STATUS <> #RESULT_SUCCESS
         THEN
           #Status := W#16#8300 OR (#receive.STATUS AND 16#00FF);
           #internalState := #STATE_IDLE;
         ELSE
           //Nothing to do, just wait here
           ;
         END_IF;

       #STATE_RECEIVE_DATA:
         // Action
         // Receive Data
         // 
         // assume job is still running
         #Status := #RESULT_JOB_RUNNING;

         #receive(EN_R := (#ownInstance = #Config.instanceLock),
                  ID := #connection.ID,
                  LEN := DWORD_TO_UINT(WORD_TO_DWORD(SWAP(UINT_TO_WORD(#receiveBuffer.Header.Length)))),
                  DATA := #receiveBuffer.Data);

         // Transition
         // Header received --> STATE_RECEIVE_DATA
         // Invalid Data --> IDLE
         // Error --> INIT
         IF #receive.NDR OR #receive.STATUS = #RESULT_SUCCESS THEN
           // Decode Response
           // 
           #currentResponse := SWAP(#receiveBuffer.Header.Command);

           //the Context will be a combination out of the own instance identifier
           //and a sequence number
           #receivedInstance := DWORD_TO_DINT(SHL(IN := USINT_TO_DWORD(#receiveBuffer.Header.Context[4]), N := 24) OR
                                              SHL(IN := USINT_TO_DWORD(#receiveBuffer.Header.Context[3]), N := 16) OR
                                              SHL(IN := USINT_TO_DWORD(#receiveBuffer.Header.Context[2]), N := 8) OR
                                              USINT_TO_DWORD(#receiveBuffer.Header.Context[1]));

           #receivedSequence := DWORD_TO_DINT(SHL(IN := USINT_TO_DWORD(#receiveBuffer.Header.Context[8]), N := 24) OR
                                              SHL(IN := USINT_TO_DWORD(#receiveBuffer.Header.Context[7]), N := 16) OR
                                              SHL(IN := USINT_TO_DWORD(#receiveBuffer.Header.Context[6]), N := 8) OR
                                              USINT_TO_DWORD(#receiveBuffer.Header.Context[5]));

           IF #currentResponse = #EIP_CMD_REG_SESSION THEN
             //Response to RegisterSession received
             // retrieve the SessionID (SessionHandle)
             IF #receiveBuffer.Header.Status = #EIP_STATUS_OK THEN
               #Config.currentSessionID := DWORD_TO_UDINT(SWAP(UDINT_TO_DWORD(#receiveBuffer.Header.SessionHandle)));
               #Status := #RESULT_SUCCESS;

             ELSE
               // inform the user about it
               //
               #Status := W#16#7100 OR DWORD_TO_WORD((SHR(IN := UDINT_TO_DWORD(#receiveBuffer.Header.Status), N := 24)));

               //Cleaning up internal information and
               //gracefully disconnect
               IF #Config.currentSessionID = 0 THEN
                 // a previous session hasn't been established --> only disconnecting
                 #internalState := #STATE_DISCONNECTING;
               ELSE
                 // previous session existed (somehow) --> unregister before disconnecting
                 #internalState := #STATE_UNREGISTER_SESSION;
               END_IF;
             END_IF;

           ELSIF #currentResponse = #EIP_CMD_SEND_RR THEN
             //Response to Send RR Data received
             // determine Status of transmission
             // retrieve TagValue and DataType
             IF #receiveBuffer.Header.Status = #EIP_STATUS_OK THEN
               #itemLength := WORD_TO_INT(SHL(IN := USINT_TO_WORD(#receiveBuffer.Data[16]), N := 8) OR USINT_TO_WORD(#receiveBuffer.Data[15]));
               #currentCIPService := USINT_TO_BYTE(#receiveBuffer.Data[17]);
               IF #currentCIPService = (#CIP_SRV_TABLEWRITE OR 16#80) AND
                 #receivedInstance = #ownInstance AND
                 #receivedSequence = #ownSequence
               THEN
                 #ownSequence := #ownSequence + 1;

                 IF #receiveBuffer.Data[19] = #CIP_GENSTS_SUCCESS THEN
                   #Status := #RESULT_SUCCESS;
                   #Done := TRUE;

                 ELSIF #receiveBuffer.Data[19] = #CIP_GENSTS_PATH_DEST_UNKNOWN OR
                       #receiveBuffer.Data[19] = #CIP_GENSTS_PATH_SEG_ERROR
                 THEN
                   // throw warning
                   #Status := W#16#7200 OR USINT_TO_BYTE(#receiveBuffer.Data[19]);

                 ELSIF #receiveBuffer.Data[19] = #CIP_GENSTS_GENERIC THEN
                   #Status := W#16#7300 OR USINT_TO_BYTE(#receiveBuffer.Data[21]);
                 ELSE
                   // throw warning
                   #Status := W#16#72FF;  //Unknown error code
                 END_IF;
               ELSIF #currentCIPService = (#CIP_SRV_TABLEWRITE_FRAG OR 16#80) THEN
                 #Status := W#16#7300 OR USINT_TO_BYTE(#receiveBuffer.Data[19]);

               ELSE
                 // throw warning
                 //   unexpected answer from host - ignoring it
                 #Status := W#16#8A00 OR #currentCIPService;
               END_IF;

             ELSE
               // inform the user about it
               //
               #Status := W#16#7100 OR DWORD_TO_WORD((SHR(IN := UDINT_TO_DWORD(#receiveBuffer.Header.Status), N := 24)));

               //Cleaning up internal information and
               //gracefully disconnect
               IF #Config.currentSessionID = 0 THEN
                 // a previous session hasn't been established --> only disconnecting
                 #internalState := #STATE_DISCONNECTING;
               ELSE
                 // previous session existed (somehow) --> unregister before disconnecting
                 #internalState := #STATE_UNREGISTER_SESSION;
               END_IF;
             END_IF;
           ELSE
             //Unknown/ Unhandled Response received
             //  ignoring it
             #Status := W#16#8B00 OR #currentResponse;
             //#Config.currentSessionID := 0;
             //#internalState := #STATE_DISCONNECTING;
           END_IF;

           #receiveBuffer.Header.Length := 0;

           //Unlocking MuteEx
           #Config.instanceLock := 0;

           #internalState := #STATE_IDLE;

         ELSIF #receive.STATUS <> #RESULT_IDLE AND
           #receive.STATUS <> #RESULT_JOB_RUNNING AND
           #receive.STATUS <> #RESULT_JOB_START AND
           #receive.STATUS <> #RESULT_SUCCESS
         THEN
           #Status := W#16#8300 OR (#receive.STATUS AND 16#00FF);
           #internalState := #STATE_IDLE;
         ELSE
           ;
         END_IF;

       #STATE_UNREGISTER_SESSION:
         IF #Config.references = 1 THEN

           #sendBuffer.Header.Command := SWAP(#EIP_CMD_UNREG_SESSION);   //Command is RegisterSession (16#66)
           #sendBuffer.Header.Length := WORD_TO_UINT(SWAP(IN := UDINT_TO_WORD(#send.LEN - #EIP_HEADER_LENGTH)));    //Length of Data is 4 Bytes
           #sendBuffer.Header.SessionHandle := DWORD_TO_UDINT(SWAP(UDINT_TO_DWORD(#Config.currentSessionID)));
           #sendBuffer.Header.Status := 0;
           #sendBuffer.Header.Options := 0;
           //the Context will be a combination out of the own instance identifier
           //and a sequence number
           #sendBuffer.Header.Context[1] := DWORD_TO_USINT(DINT_TO_DWORD(#ownInstance) AND DW#16#000000FF);
           #sendBuffer.Header.Context[2] := DWORD_TO_USINT(SHR(IN := DINT_TO_DWORD(#ownInstance), N := 8) AND DW#16#000000FF);
           #sendBuffer.Header.Context[3] := DWORD_TO_USINT(SHR(IN := DINT_TO_DWORD(#ownInstance), N := 16) AND DW#16#000000FF);
           #sendBuffer.Header.Context[4] := DWORD_TO_USINT(SHR(IN := DINT_TO_DWORD(#ownInstance), N := 24) AND DW#16#000000FF);
           #sendBuffer.Header.Context[5] := DWORD_TO_USINT(DINT_TO_DWORD(#ownSequence) AND DW#16#000000FF);
           #sendBuffer.Header.Context[6] := DWORD_TO_USINT(SHR(IN := DINT_TO_DWORD(#ownSequence), N := 8) AND DW#16#000000FF);
           #sendBuffer.Header.Context[7] := DWORD_TO_USINT(SHR(IN := DINT_TO_DWORD(#ownSequence), N := 16) AND DW#16#000000FF);
           #sendBuffer.Header.Context[8] := DWORD_TO_USINT(SHR(IN := DINT_TO_DWORD(#ownSequence), N := 24) AND DW#16#000000FF);
           #sendBuffer.Data[1] := 16#00;

           //Checking the MuteEx
           IF #Config.instanceLock = 0 OR
             #Config.instanceLock = #ownInstance
           THEN
             //Locking the MutEx
             #Config.instanceLock := #ownInstance;
             #send.LEN := #EIP_HEADER_LENGTH;
             #send.REQ := TRUE;
             // Action
             // 

             #send(ID := #connection.ID,
                   DATA := #sendBuffer);

             // Transition
             //
             #internalState := #STATE_UNREGISTERING;
             #Config.references := #Config.references - 1;
           ELSE
             IF #Config.instanceLock = #ownInstance THEN
               #Config.instanceLock := 0;
             END_IF;
           END_IF;
         ELSE
           IF #Config.references > 1 THEN
             #Config.references := #Config.references - 1;
           END_IF;
           #internalState := #STATE_POWER_OFF;
         END_IF;

       #STATE_UNREGISTERING:
         // Action
         // 

         #send(ID := #connection.ID,
               DATA := #sendBuffer);

         // Transition
         //
         IF #send.STATUS = #RESULT_JOB_START THEN
           ;
         ELSIF #send.STATUS = #RESULT_JOB_RUNNING THEN
           #send.REQ := FALSE;

         ELSIF #send.STATUS = #RESULT_IDLE THEN
           #send.REQ := NOT #send.REQ; 

         ELSIF #send.STATUS = #RESULT_SUCCESS THEN
           #send.REQ := FALSE;
           #internalState := #STATE_DISCONNECTING;
           //Unlocking MuteEx
           #Config.instanceLock := 0;

         ELSE
           // Throw error !
           //   Error from Sending
           #Status := W#16#8200 OR (#send.STATUS AND 16#00FF);
           #send.REQ := FALSE;
           #internalState := #STATE_DISCONNECTING;
         END_IF;

       #STATE_DISCONNECTING:

         IF #disconnect.STATUS = #RESULT_JOB_START THEN
           #connectionStatus.isConnected := FALSE;
           #connectionStatus.isDisconnecting := TRUE;

         ELSIF #disconnect.STATUS = #RESULT_IDLE THEN
           #connectionStatus.isDisconnecting := TRUE;
           #disconnect.REQ := NOT #disconnect.REQ;

         ELSIF #disconnect.STATUS = #RESULT_JOB_RUNNING THEN
           #disconnect.REQ := FALSE;

         ELSIF #disconnect.STATUS = #RESULT_JOB_NOT_REQUIRED OR
           #disconnect.STATUS = #RESULT_SUCCESS
         THEN
           #disconnect.REQ := FALSE;
           #connectionStatus.isConnected := FALSE;
           #connectionStatus.isDisconnecting := FALSE;
           #connectionStatus.isDisconnected := TRUE;
           #connectionStatus.hasReceivedData := FALSE;
           #connectionStatus.hasReceivedHeader := FALSE;
           //#Config.currentSessionID := 0;
           #ownInstance := 0;
           #ownSequence := 0;
           #Config.connID := 0;

           #internalState := #STATE_IDLE;
         ELSE
           // Throw error !
           //   Error from disconnecting
           #Status := W#16#8400 OR (#disconnect.STATUS AND 16#00FF);
           #disconnect.REQ := FALSE;
           #connectionStatus.isConnected := FALSE;
           #connectionStatus.isDisconnecting := FALSE;
           #connectionStatus.isDisconnected := TRUE;
           #connectionStatus.hasReceivedData := FALSE;
           #connectionStatus.hasReceivedHeader := FALSE;

           //#Config.currentSessionID := 0;
           #ownInstance := 0;
           #ownSequence := 0;

           #internalState := #STATE_IDLE;
         END_IF;
       ELSE
         // Throw error !
         //   unknown internal state        
         #Status := W#16#8C00 OR (UINT_TO_WORD(#internalState) AND W#16#00FF);
     END_CASE;
   END_IF;

   #previousRequest := #REQ;
   #EnabledJ := #Enable;

   // Diagnose the connection

   #diag(ID := #connection.ID,
         RESULT := #diagStatus);

   IF #diag.STATUS = #RESULT_SUCCESS THEN
     #diag.REQ := FALSE;
     #Established := (#diagStatus.State = B#16#04);
     #Connecting := (#diagStatus.State = B#16#02) OR (#diagStatus.State = B#16#01);
   ELSIF #diag.STATUS = #RESULT_IDLE OR #diag.STATUS = #RESULT_JOB_START THEN
     #diag.REQ := TRUE;
   ELSIF #diag.STATUS = #RESULT_JOB_RUNNING THEN
     #diag.REQ := FALSE;
   ELSE
     #diag.REQ := FALSE;
     #Established := FALSE;
     #Connecting := FALSE;
   END_IF;
END_FUNCTION_BLOCK

FUNCTION_BLOCK "GET_R"   // FB7, SCL
{ S7_Optimized_Access := 'TRUE' }
VERSION : 0.1
   VAR_INPUT
      Enable : Bool;   // [TRUE| FALSE] TRUE signal keeps the block in PowerOff state
      REQ : Bool;   // [TRUE |FALSE] rising edge triggers a read request
      InterfaceId : Hw_Interface;   // [1..] InterfaceID of the used interface
      IPv4 : IP_V4;   // [IP v4 address] IP address of the remote rack
      Slot : Int;   // [-1..16] Slot the addressed CPU is located; -1 if directly connected
   END_VAR
   VAR_OUTPUT
      Status : Word;   // [Enum] status information
      NewData : Bool;   // [TRUE | FALSE] TRUE signal is a one shot signal indicating the receiption of the requested data
      Connecting : Bool;   // [TRUE | FALSE] TRUE signal indicates the establishment of the connection
      Established : Bool;   // [TRUE | FALSE] TRUE indicates an established connection
   END_VAR
   VAR_IN_OUT
      Config : "RockwellConfig";
      Tag : "RockwellTag";   // [RockwelTag] datatype containing the tagname, value and data type
      Value : Variant;
   END_VAR
   VAR
      internalState : UInt;   // [Enum] contains the internal state information
      connect : TCON;
      disconnect : TDISCON;
      send : TSEND;
      receive : TRCV;
      diag : T_DIAG;
      connection : TCON_IP_v4;
      sendBuffer : Struct
         Header : Struct
            Command : Word;   // Encapsulation command
            Length : UInt;   // Length, in bytes, of the command specific data portion of the message
            SessionHandle : UDInt;   // Session identification
            Status : UDInt;   // Status code
            Context : Array[1..8] of USInt;   // Information pertinien only to the sender of an encapsulation command
            Options : UDInt;
         END_STRUCT;
         Data : Array[1..508] of USInt;
      END_STRUCT;
      receiveBuffer : Struct
         Header : Struct
            Command : Word;   // Encapsulation command
            Length : UInt;   // Length, in bytes, of the command specific data portion of the message
            SessionHandle : UDInt;   // Session identification
            Status : UDInt;   // Status code
            Context : Array[1..8] of USInt;   // Information pertinien only to the sender of an encapsulation command
            Options : UDInt;
         END_STRUCT;
         Data : Array[1..508] of USInt;
      END_STRUCT;
      currentResponse : Word;
      connectionStatus : Struct
         isDisconnected : Bool;
         isDisconnecting : Bool;
         isConnecting : Bool;
         isConnected : Bool;
         hasReceivedData : Bool;
         hasReceivedHeader : Bool;
      END_STRUCT;
      indexTag : Int := 0;
      currentCIPService : Byte;
      previousRequest : Bool;
      EnabledJ : Bool;
      ownInstance : DInt;
      ownSequence : DInt;
      diagStatus : TDiag_StatusExt;
      randomGenerator : Struct   // [STRUCT] used to realize a pseudo random number
         m_w : DInt;
         m_z : DInt;
         Val : DInt;
         currentTime : DTL;
         currentMilliSeconds : DInt;
      END_STRUCT;
   END_VAR
   VAR_TEMP
      indexTagName : DInt;
      result : Int;
      itemLength : DInt;   // contains the Length of the EIP packet
      overallLength : DInt;   // contains the Length of the EIP packet
      tagNameLength : DInt;   // contains the Length of the Tagname (in WORDS)
      unconnectedDataItemLength : DInt;   // contains the Length of the unconnected data item
      baseIndexOuterCIPMessage : DInt;   // contains the base index to the beginning of the outer CIP message
      baseIndexInnerCIPMessage : DInt;   // contains the base index to the beginning of the inner CIP message
      receivedInstance : DInt;
      receivedSequence : DInt;
      receivedType : Word;
      valueIndex : Int;
      receivedValue : Struct
         Boolean : Bool;
         Short : SInt;
         Integer : Int;
         Double : DInt;
         Float : Real;
      END_STRUCT;
   END_VAR
   VAR CONSTANT
      EIP_VENDOR_ID : Word := 1251;   // EtherNet/IP vendor ID 'Siemens AG'
      EIP_HEADER_LENGTH : UInt := 24;   // EtherNet/IP Encapsulation Header length is 24 bytes
      EIP_PORT : Word := 44818;   // EtherNet/IP standard port is 44818 (0xAF12)
      RESULT_SUCCESS : Word := 16#0000;
      RESULT_IDLE : Word := 16#7000;
      RESULT_JOB_START : Word := 16#7001;
      RESULT_JOB_RUNNING : Word := 16#7002;
      RESULT_JOB_NOT_REQUIRED : Word := 16#80A3;
      RESULT_MORE_AVAIL : Word := 16#80B1;
      RESULT_REUSED_ID : Word := 16#8085;
      EIP_STATUS_OK : UDInt := 0;   // EIP Status OK
      EIP_STATUS_TOOMANY_SESSIONS : UDInt := 16#01000000;   // EIP Status "more than 1 active session on the same TCP connection"
      EIP_STATUS_OUTOFRESSOURCES : UDInt := 16#02000000;   // EIP Status "does not have sufficient resources"
      EIP_STATUS_INVALID_SESSION_ID : UDInt := 16#64000000;   // EIP Status "Invalid Session ID"
      EIP_STATUS_PROTOCOL_ERROR : UDInt := 16#69000000;   // EIP Status "Protocol Version or Options mismatches"
      EIP_CMD_REG_SESSION : Word := 16#0065;   // EtherNet/IP Encapsulation Command "Register Session"
      EIP_CMD_UNREG_SESSION : Word := 16#0066;   // EtherNet/IP Encapsulation Command "Unregister Session"
      EIP_CMD_SEND_RR : Word := 16#006F;   // EtherNet/IP Encapsulation Command "Send RR Data"
      CIP_SRV_TABLEREAD : Byte := 16#4C;   // CIP Service Data Table Read
      CIP_SRV_TABLEWRITE : Byte := 16#4D;   // CIP Service Data Table Write
      CIP_SRV_TABLEREAD_FRAG : Byte := 16#52;   // CIP Service Fragmented Data Table Read
      CIP_SRV_TABLEWRITE_FRAG : Byte := 16#53;   // CIP Service Fragmented Data Table Write
      CIP_SRV_UNCONNECTED_SEND : Byte := 16#52;   // CIP Service Unconnected Send Data
      STATE_IDLE : UInt := 1;
      STATE_INIT : UInt := 2;
      STATE_CONNECTING : UInt := 3;
      STATE_DISCONNECTING : UInt := 4;
      STATE_SENDING : UInt := 5;
      STATE_REGISTER_SESSION : UInt := 6;
      STATE_UNREGISTER_SESSION : UInt := 7;
      STATE_REGISTERING : UInt := 8;
      STATE_UNREGISTERING : UInt := 9;
      STATE_REGISTERED : UInt := 10;
      STATE_SEND : UInt := 11;
      STATE_RECEIVE_HEADER : UInt := 12;
      STATE_RECEIVE_DATA : UInt := 13;
      STATE_POWER_OFF : UInt := 0;
      DT_BOOLEAN_ATOMIC : USInt := 16#C1;
      DT_SINT_ATOMIC : USInt := 16#C2;
      DT_INT_ATOMIC : USInt := 16#C3;
      DT_DINT_ATOMIC : USInt := 16#C4;
      DT_FLOAT_ATOMIC : USInt := 16#CA;
      CIP_PATH_SEG_TYPE_CLASS : USInt := 16#20;
      CIP_PATH_SEG_TYPE_INSTANCE : USInt := 16#24;
      CIP_PATH_SEG_TYPE_ANSI : USInt := 16#91;
      CIP_PATH_SEG_TYPE_PORT : USInt := 16#01;
      CIP_ROUTE_SEG_LENGTH : Int := 4;
      CIP_ROUTE_PATH_LENGTH : Int := 1;
      CIP_TABLEREAD_LENGTH : Int := 6;
      CIP_TABLEWRITE_LENGTH : Int := 4;
      CIP_UCSEND_HEADER_LENGTH : Int := 4;
      CIP_UCSEND_SEG_LENGTH : Int := 6;
      EIP_CMD_SEND_RR_SEG_LENGTH : Int := 16;
      CON_TYPE_TCP_V2 : USInt := 17;   // TCP connection for TCON_PARAM descriptor
      CON_TYPE_TCP_V4 : Byte := 11;   // TCP connection for TCON_IP_V4 descriptor
      CIP_GENSTS_SUCCESS : USInt := 16#00;
      CIP_GENSTS_PATH_SEG_ERROR : USInt := 16#04;
      CIP_GENSTS_PATH_DEST_UNKNOWN : USInt := 16#05;
      CIP_GENSTS_PARTIAL : USInt := 16#06;
      CIP_GENSTS_NOT_ENOUGH_DATA : USInt := 16#13;
      CIP_GENSTS_PATH_SIZE_MISMATCH : USInt := 16#26;
      CIP_GENSTS_DOESNT_EXIST : USInt := 16#16;
      CIP_GENSTS_GENERIC : USInt := 16#FF;
      CIP_SRVSTS_RANGE_EXCEED : UInt := 16#2105;
   END_VAR
BEGIN
   //=============================================================================
   // Siemens AG
   // (c)Copyright 2016 All Rights Reserved
   //-----------------------------------------------------------------------------
   // Library: PutGet_Rockwell
   // Tested with: 1511-1 PN V1.8.3 and ControlLogix/Compactlogix V26
   // Engineering: TIA Portal V13 SP1 Upd 9
   // Restrictions: look into pdf
   // Requirements: S7-1500 V1.8.3
   // Functionality: Get Put Values from to Rockwell CPU
   //-----------------------------------------------------------------------------
   // Change log table:
   // Version  Date            Expert in charge        Changes applied
   // 01.00.00 12.07.2016      Scheel                  initial version 
   // 01.00.01 22.07.2016      Scheel                  feat: add diagnostics and
   //                                                        indicators
   // 01.00.02 28.07.2016      Scheel                  style: remove duplicate
   //                                                         code segments
   // 01.00.04 19.10.2016      Scheel                  fix: connect will be
   //                                                       retriggered, when idle
   //                                                  refac: change of IP address
   //                                                         datatype to IP_V4
   //                                                  feat: add recognition of
   //                                                        CIP specific status
   //=============================================================================
   //

   //#########################################################################################
   // Pseudo Random number generator
   //
   //  This Random number function generator is based on multiplication and
   //  addition with overflow invented by George Marsaglia.
   //  The loss of information is intended.
   //  
   //  Wikipedia (https://en.wikipedia.org/wiki/Random_number_generation)
   //#########################################################################################
   //
   //Initialization of the variables using a time value as a seed
   #result := RD_SYS_T(#randomGenerator.currentTime);
   #randomGenerator.currentMilliSeconds := UDINT_TO_DINT(#randomGenerator.currentTime.NANOSECOND) / 1000000 + (USINT_TO_DINT(#randomGenerator.currentTime.SECOND) * 1000);

   IF #randomGenerator.m_w = 0 OR #randomGenerator.m_z = 0 THEN
     #randomGenerator.m_w := UDINT_TO_DINT((#randomGenerator.currentTime.NANOSECOND / 1000000)) + 2;    // using the milliseconds since the PLC has been powered on
     #randomGenerator.m_z := 13696;
   ELSE
     #randomGenerator.m_z := 36969 * DWORD_TO_DINT(DINT_TO_DWORD(#randomGenerator.m_z) AND 16#FFFF)
     + DWORD_TO_DINT(SHR(IN := DINT_TO_DWORD(#randomGenerator.m_z), N := 16));
     #randomGenerator.m_w := 18000 * DWORD_TO_DINT(DINT_TO_DWORD(#randomGenerator.m_w) AND 16#FFFF)
     + DWORD_TO_DINT(SHR(IN := DINT_TO_DWORD(#randomGenerator.m_w), N := 16));
     #randomGenerator.Val := DWORD_TO_DINT(SHL(IN := DINT_TO_DWORD(#randomGenerator.m_z), N := 16)) + #randomGenerator.m_w;  // 32-bit result */    
   END_IF;

   //assume idle state
   #Status := #RESULT_IDLE;
   #NewData := FALSE;

   #connect(ID := #connection.ID,
            CONNECT := #connection);

   #disconnect(ID := #connection.ID);


   IF NOT #Enable AND #EnabledJ THEN
     // Complete Restart detected 
     //
     #internalState := #STATE_UNREGISTER_SESSION;

   ELSIF #Enable AND NOT #EnabledJ THEN  
     #internalState := #STATE_INIT;

   ELSE
     // Regular operation
     //
     CASE #internalState OF
       #STATE_POWER_OFF:
         //Preset the TCP connection information
         //
         IF #Config.connID = 0 THEN
           #Config.connID := DWORD_TO_WORD(DINT_TO_DWORD((#randomGenerator.Val MOD 2048) + 2048));
         END_IF;
         #connection.ID := #Config.connID;

         // only usable in S7-1500 or S7-1200 V4.x
         // 
         #connection.ConnectionType := #CON_TYPE_TCP_V4;           //TCP connection
         #connection.InterfaceId := #InterfaceId;
         #connection.ActiveEstablished := TRUE;             //active connection (Client)

         #connection.RemoteAddress := #IPv4;

         #connection.RemotePort := WORD_TO_UINT(#EIP_PORT);

         // #connection.CONNECTION_TYPE := #CON_TYPE_TCP_V2;      //TCP connection
         // #connection.LOCAL_DEVICE_ID := WORD_TO_USINT(#InterfaceId);
         // #connection.ACTIVE_EST := TRUE;                //active connection (Client)

         // #connection.REM_STADDR_LEN := 4;
         // #connection.REM_STADDR[1] := BYTE_TO_USINT(#IPv4[1]);
         // #connection.REM_STADDR[2] := BYTE_TO_USINT(#IPv4[2]);
         // #connection.REM_STADDR[3] := BYTE_TO_USINT(#IPv4[3]);
         // #connection.REM_STADDR[4] := BYTE_TO_USINT(#IPv4[4]);

         // #connection.REM_TSAP_ID_LEN := 2;
         // #connection.REM_TSAP_ID[1] := WORD_TO_BYTE(SHR(IN := #EIP_PORT, N := 8));
         // #connection.REM_TSAP_ID[2] := WORD_TO_BYTE(#EIP_PORT AND W#16#FF);

         #ownInstance := 0;
         #ownSequence := 0;

         #internalState := #STATE_IDLE;

       #STATE_IDLE:

         // Action
         //
         #NewData := FALSE;

         // Transition 
         //IF NOT #connectionStatus.isConnected THEN
         //  #internalState := #STATE_INIT;
         IF #connectionStatus.isConnected AND #REQ AND NOT #previousRequest AND #Enable THEN
           #internalState := #STATE_SENDING;
           #Status := #RESULT_JOB_START;
         END_IF;


       #STATE_INIT:
         //Preset the TCP connection information
         //
         IF #Config.connID = 0 THEN
           #Config.connID := DWORD_TO_WORD(DINT_TO_DWORD((#randomGenerator.Val MOD 2048) + 2048));
         END_IF;
         #connection.ID := #Config.connID;

         //Inserting Semaphore checking
         //
         //  Only issue a new connect, when there is no one is referencing the connection already
         //  Otherwise just skip that step and use the established connection
         //  

         IF #Config.references = 0 THEN
           // only usable in S7-1500 or S7-1200 V4.x
           // 
           #connection.ConnectionType := #CON_TYPE_TCP_V4;    //TCP connection
           #connection.InterfaceId := #InterfaceId;
           #connection.ActiveEstablished := TRUE;             //active connection (Client)

           #connection.RemoteAddress := #IPv4;

           #connection.RemotePort := WORD_TO_UINT(#EIP_PORT);

           // #connection.CONNECTION_TYPE := #CON_TYPE_TCP_V2;      //TCP connection
           // #connection.LOCAL_DEVICE_ID := WORD_TO_USINT(#InterfaceId);
           // #connection.ACTIVE_EST := TRUE;                //active connection (Client)

           // #connection.REM_STADDR_LEN := 4;
           // #connection.REM_STADDR[1] := BYTE_TO_USINT(#IPv4[1]);
           // #connection.REM_STADDR[2] := BYTE_TO_USINT(#IPv4[2]);
           // #connection.REM_STADDR[3] := BYTE_TO_USINT(#IPv4[3]);
           // #connection.REM_STADDR[4] := BYTE_TO_USINT(#IPv4[4]);

           // #connection.REM_TSAP_ID_LEN := 2;
           // #connection.REM_TSAP_ID[1] := WORD_TO_BYTE(SHR(IN := #EIP_PORT, N := 8));
           // #connection.REM_TSAP_ID[2] := WORD_TO_BYTE(          #EIP_PORT AND W#16#FF);


           //No connection established yet
           //  issue a new request
           #connect.REQ := TRUE;
           #internalState := #STATE_CONNECTING;
         ELSE
           #internalState := #STATE_IDLE;
           #connectionStatus.isConnected := TRUE;
         END_IF;
         #Config.references := #Config.references + 1;

         //Remember the currently active instance reference as my own instance identifier
         //  and reset the Sequence counter
         #ownInstance := #Config.references;
         #ownSequence := 0;

       #STATE_CONNECTING:

         IF #connect.STATUS = #RESULT_JOB_START THEN
           #connectionStatus.isConnecting := TRUE;

         ELSIF #connect.STATUS = #RESULT_IDLE THEN
           #connect.REQ := NOT #connect.REQ;

         ELSIF #connect.STATUS = #RESULT_JOB_RUNNING THEN
           #connect.REQ := FALSE;

         ELSIF #connect.STATUS = #RESULT_JOB_NOT_REQUIRED OR
               #connect.STATUS = #RESULT_SUCCESS 
         THEN
           #connect.REQ := FALSE;
           #connectionStatus.isConnecting := FALSE;
           #connectionStatus.isConnected := TRUE;
           #connectionStatus.isDisconnected := FALSE;

           #internalState := #STATE_REGISTER_SESSION;

         ELSE
           // Throw error !
           //   Error in connect
           #Status := W#16#8100 OR (#connect.STATUS AND 16#00FF);   //Error in connecting
           #connect.REQ := FALSE;
           #internalState := #STATE_DISCONNECTING;
         END_IF;

       #STATE_REGISTER_SESSION:

         #sendBuffer.Header.Command := SWAP(#EIP_CMD_REG_SESSION);                            //Command is RegisterSession (16#65)
         #sendBuffer.Header.Length  := WORD_TO_UINT(SWAP(IN := UDINT_TO_WORD(4)));            //Length of Data is 4 Bytes
         #sendBuffer.Header.SessionHandle := 0;
         #sendBuffer.Header.Status := 0;
         #sendBuffer.Header.Options := 0;
         //the Context will be a combination out of the own instance identifier
         //and a sequence number
         #sendBuffer.Header.Context[1] := DWORD_TO_USINT(        DINT_TO_DWORD(#ownInstance)        AND DW#16#000000FF);
         #sendBuffer.Header.Context[2] := DWORD_TO_USINT(SHR(IN:=DINT_TO_DWORD(#ownInstance),N:= 8) AND DW#16#000000FF);
         #sendBuffer.Header.Context[3] := DWORD_TO_USINT(SHR(IN:=DINT_TO_DWORD(#ownInstance),N:=16) AND DW#16#000000FF);
         #sendBuffer.Header.Context[4] := DWORD_TO_USINT(SHR(IN:=DINT_TO_DWORD(#ownInstance),N:=24) AND DW#16#000000FF);
         #sendBuffer.Header.Context[5] := DWORD_TO_USINT(        DINT_TO_DWORD(#ownSequence)        AND DW#16#000000FF);
         #sendBuffer.Header.Context[6] := DWORD_TO_USINT(SHR(IN:=DINT_TO_DWORD(#ownSequence),N:= 8) AND DW#16#000000FF);
         #sendBuffer.Header.Context[7] := DWORD_TO_USINT(SHR(IN:=DINT_TO_DWORD(#ownSequence),N:=16) AND DW#16#000000FF);
         #sendBuffer.Header.Context[8] := DWORD_TO_USINT(SHR(IN:=DINT_TO_DWORD(#ownSequence),N:=24) AND DW#16#000000FF);
         #sendBuffer.Data[1] := 16#01;                                 //Protocol Version V1.0

         //Checking the MuteEx
         IF #Config.instanceLock = 0 OR
           #Config.instanceLock = #ownInstance
         THEN
           //allowed to utilize, since instanceLock is either 0 or ownInstance
           #send(ID := #connection.ID,
                 DATA := #sendBuffer);

           //Locking the MutEx
           #Config.instanceLock := #ownInstance;
           #send.LEN := #EIP_HEADER_LENGTH + 4;
           #send.REQ := TRUE;

           #internalState := #STATE_REGISTERING;
         ELSE
           ;
         END_IF;

       #STATE_REGISTERING:
         // Action
         // 

         //allowed to utilize, since instanceLock is either 0 or ownInstance
         #send(ID := #connection.ID,
               DATA := #sendBuffer);

         // Transition
         // 
         IF #send.STATUS = #RESULT_JOB_START THEN
           ;
         ELSIF #send.STATUS = #RESULT_JOB_RUNNING THEN
           #send.REQ := FALSE;

         ELSIF #send.STATUS = #RESULT_IDLE THEN
           #send.REQ := NOT #send.REQ;

         ELSIF #send.STATUS = #RESULT_SUCCESS THEN
           #send.REQ := FALSE;
           #internalState := #STATE_RECEIVE_HEADER;
         ELSE
           // Throw error !
           //   in Registering
           #Status := W#16#8200 OR (#send.STATUS AND 16#00FF);   //Error in sending
           #send.REQ := FALSE;
           #internalState := #STATE_DISCONNECTING;
         END_IF;

       #STATE_SENDING:
         #sendBuffer.Header.Command := SWAP(#EIP_CMD_SEND_RR);                                                 //Command is SendRRData (16#6F)
         //
         // overall Message length depends on the packet content and is therefore assigned later
         //
         #sendBuffer.Header.SessionHandle := DWORD_TO_UDINT(SWAP(UDINT_TO_DWORD(#Config.currentSessionID)));;
         #sendBuffer.Header.Status := 0;
         #sendBuffer.Header.Options := 0;
         //the Context will be a combination out of the own instance identifier
         //and a sequence number
         #sendBuffer.Header.Context[1] := DWORD_TO_USINT(DINT_TO_DWORD(#ownInstance) AND DW#16#000000FF);
         #sendBuffer.Header.Context[2] := DWORD_TO_USINT(SHR(IN := DINT_TO_DWORD(#ownInstance), N := 8) AND DW#16#000000FF);
         #sendBuffer.Header.Context[3] := DWORD_TO_USINT(SHR(IN := DINT_TO_DWORD(#ownInstance), N := 16) AND DW#16#000000FF);
         #sendBuffer.Header.Context[4] := DWORD_TO_USINT(SHR(IN := DINT_TO_DWORD(#ownInstance), N := 24) AND DW#16#000000FF);
         #sendBuffer.Header.Context[5] := DWORD_TO_USINT(DINT_TO_DWORD(#ownSequence) AND DW#16#000000FF);
         #sendBuffer.Header.Context[6] := DWORD_TO_USINT(SHR(IN := DINT_TO_DWORD(#ownSequence), N := 8) AND DW#16#000000FF);
         #sendBuffer.Header.Context[7] := DWORD_TO_USINT(SHR(IN := DINT_TO_DWORD(#ownSequence), N := 16) AND DW#16#000000FF);
         #sendBuffer.Header.Context[8] := DWORD_TO_USINT(SHR(IN := DINT_TO_DWORD(#ownSequence), N := 24) AND DW#16#000000FF);
         //CIP specific data
         #sendBuffer.Data[1] := 16#0;                                 //CIP Interface handle
         #sendBuffer.Data[2] := 16#0;
         #sendBuffer.Data[3] := 16#0;
         #sendBuffer.Data[4] := 16#0;

         #sendBuffer.Data[5] := 16#0;                                  //Timeout
         #sendBuffer.Data[6] := 16#0;

         #sendBuffer.Data[7] := 16#2;                                  //Items
         #sendBuffer.Data[8] := 16#0;

         #sendBuffer.Data[9] := 16#0;                                  //Null address item
         #sendBuffer.Data[10] := 16#0;
         #sendBuffer.Data[11] := 16#0;                                  //Null address item Length = 0
         #sendBuffer.Data[12] := 16#0;

         #sendBuffer.Data[13] := 16#B2;                                  //Unconnected data item
         #sendBuffer.Data[14] := 16#0;
         //Item Length needs to be added, but since that depends on the content,
         //it will will be assigned later. It occupies 2 Bytes, thus the outer CIP Message 
         //starts at offset 17 into the Data (1 based counting)
         //
         #baseIndexOuterCIPMessage := 17;

         //CIP Message
         //  here a decision needs to be made
         //  In case Slot is -1 a direct connection is assumed, such as for a CompactLogix, this means no
         //  further route segments are necessary
         //  In case Slot is anywhere between 0 and 16 a route segment is required, since the CPU is not
         //  identical to the ethernet interface, as in a ControlLogix L5, L6, L7 series system

         //Length of the following Path segment depends only on the length of the Tagname measured in WORDS
         // plus 1 WORD for the segment encoding information
         // 
         #tagNameLength := ((LEN(#Tag."Name") + 1) / 2) * 2;

         //
         //  Prelude
         //
         //In case the slot information is negative (-1) there is no additional path segment
         //Any other slot value requires routing information, which need to be added
         //  this means the preparation of offsets and header needs to be done, before
         //  the common part of copying the value to the packet can take place
         IF #Slot = -1 THEN
           //directly connected (onboard) Ethernet interface
           //
           #baseIndexInnerCIPMessage := #baseIndexOuterCIPMessage;

         ELSE
           //not directly connected (through external) Ethernet interface
           //
           //  preparing offsets for length calculation as well as header
           //  There is a 10 byte segment before the tag value segment
           #baseIndexInnerCIPMessage := #baseIndexOuterCIPMessage + 10;

           #sendBuffer.Data[#baseIndexOuterCIPMessage] :=  BYTE_TO_USINT(#CIP_SRV_UNCONNECTED_SEND);  //CIP service = UNCONNECTED_SEND_DATA = 16#52
           #sendBuffer.Data[#baseIndexOuterCIPMessage + 1] := 2;                                     //Path Size is constant 2 WORDS

           #sendBuffer.Data[#baseIndexOuterCIPMessage + 2] := #CIP_PATH_SEG_TYPE_CLASS;              //Path Type = Class Segment
           #sendBuffer.Data[#baseIndexOuterCIPMessage + 3] := 16#06;                                 //Class = ConnectionManager (16#06)

           #sendBuffer.Data[#baseIndexOuterCIPMessage + 4] := #CIP_PATH_SEG_TYPE_INSTANCE;           //Path Type = Instance Segment
           #sendBuffer.Data[#baseIndexOuterCIPMessage + 5] := 16#01;                                 //Instance =Instance 1 (16#01)

           //Encapsulated CIP Message
           //
           #sendBuffer.Data[#baseIndexOuterCIPMessage + 6] := 16#07;                                 //Priority combined with TimeTick (= 16#07)
           #sendBuffer.Data[#baseIndexOuterCIPMessage + 7] := INT_TO_USINT(233);                     //???

         END_IF;

         //
         // tag value segment
         // 

         #sendBuffer.Data[#baseIndexInnerCIPMessage] := BYTE_TO_USINT(#CIP_SRV_TABLEREAD);      //CIP service = DATA_TABLE_READ = 16#4C

         #sendBuffer.Data[#baseIndexInnerCIPMessage + 1] := DINT_TO_USINT(#tagNameLength / 2 + 1);  //Path Size
         #sendBuffer.Data[#baseIndexInnerCIPMessage + 2] := #CIP_PATH_SEG_TYPE_ANSI;            //Path Type = ANSI Extended Symbol Segment

         //Copy In

         #sendBuffer.Data[#baseIndexInnerCIPMessage + 3] := INT_TO_USINT(LEN(#Tag."Name"));   //TagName Length (bytes)
         FOR #indexTagName := 1 TO USINT_TO_INT(#sendBuffer.Data[#baseIndexInnerCIPMessage + 3]) DO
           #sendBuffer.Data[#baseIndexInnerCIPMessage + 3 + #indexTagName] := CHAR_TO_USINT(#Tag."Name"[#indexTagName]);
         END_FOR;

         //in case the tag name has an odd (uneven) length the path segment content needs to be padded to be WORD aligned
         //
         #indexTagName := #indexTagName - 1;
         IF #indexTagName MOD 2 <> 0 THEN
           #indexTagName := #indexTagName + 1;
           #sendBuffer.Data[#baseIndexInnerCIPMessage + 3 + #indexTagName] := 0;
         END_IF;

         //Command Specific information
         //

         #sendBuffer.Data[#baseIndexInnerCIPMessage + 4 + #indexTagName] := INT_TO_USINT(#Tag.Count);                  //Number of Items
         #sendBuffer.Data[#baseIndexInnerCIPMessage + 5 + #indexTagName] := WORD_TO_USINT(SHR(IN := INT_TO_WORD(#Tag.Count), N := 8) AND W#16#00FF);

         #itemLength := #tagNameLength + #CIP_TABLEREAD_LENGTH;

         //
         // Closure
         //

         IF #Slot = -1 THEN
           #unconnectedDataItemLength := #itemLength;
         ELSE
           #sendBuffer.Data[#baseIndexOuterCIPMessage + 8] := WORD_TO_USINT(DINT_TO_WORD(#itemLength));                     //Unconnected data item Length
           #sendBuffer.Data[#baseIndexOuterCIPMessage + 9] := WORD_TO_USINT(SHL(IN := DINT_TO_WORD(#itemLength), N := 8));  //Unconnected data item Length

           //Routing Information
           #sendBuffer.Data[#baseIndexInnerCIPMessage + #itemLength    ] := INT_TO_USINT(#CIP_ROUTE_PATH_LENGTH);
           #sendBuffer.Data[#baseIndexInnerCIPMessage + #itemLength + 1] := 0;

           #sendBuffer.Data[#baseIndexInnerCIPMessage + #itemLength + 2] := #CIP_PATH_SEG_TYPE_PORT;
           #sendBuffer.Data[#baseIndexInnerCIPMessage + #itemLength + 3] := INT_TO_USINT(#Slot);

           #unconnectedDataItemLength :=   #itemLength
                                         + #CIP_ROUTE_SEG_LENGTH
                                         + #CIP_UCSEND_HEADER_LENGTH
                                         + #CIP_UCSEND_SEG_LENGTH;
         END_IF;

         //Length of the unconnected data item depends on the content of the package
         //
         #sendBuffer.Data[15] := WORD_TO_USINT(DINT_TO_WORD(#unconnectedDataItemLength));                //Unconnected data item Length
         #sendBuffer.Data[16] := WORD_TO_USINT(SHL(IN:=DINT_TO_WORD(#unconnectedDataItemLength),N:=8));  //Unconnected data item Length

         #sendBuffer.Header.Length := WORD_TO_UINT(SWAP(IN := DINT_TO_WORD(#unconnectedDataItemLength + #EIP_CMD_SEND_RR_SEG_LENGTH)));    //Length of Data

         //Checking the MuteEx
         IF #Config.instanceLock = 0 OR
           #Config.instanceLock = #ownInstance
         THEN
           //Locking the MutEx
           #Config.instanceLock := #ownInstance;
           #send.LEN := DINT_TO_UINT(#EIP_HEADER_LENGTH + #unconnectedDataItemLength + #EIP_CMD_SEND_RR_SEG_LENGTH);
           #send.REQ := TRUE;

           //allowed to utilize, since instanceLock is either 0 or ownInstance
           #send(ID := #connection.ID,
                 DATA := #sendBuffer);

           #internalState := #STATE_SEND;
         ELSE
           ;
         END_IF;
         #Status := #RESULT_JOB_RUNNING;

       #STATE_SEND:
         // Action
         // 
         // assume job is still running
         #Status := #RESULT_JOB_RUNNING;

         #send(ID := #connection.ID,
               DATA := #sendBuffer);

         // Transition
         //
         IF #send.STATUS = #RESULT_JOB_START THEN
           ;
         ELSIF #send.STATUS = #RESULT_IDLE THEN
           #send.REQ := NOT #send.REQ;

         ELSIF #send.STATUS = #RESULT_JOB_RUNNING THEN
           #send.REQ := FALSE;

         ELSIF #send.STATUS = #RESULT_SUCCESS THEN
           #send.REQ := FALSE;
           #internalState := #STATE_RECEIVE_HEADER;
         ELSE
           // Throw error !
           // 
           #Status := W#16#8200 OR (#send.STATUS AND 16#00FF);
           #send.REQ := FALSE;
           #internalState := #STATE_DISCONNECTING;
         END_IF;


       #STATE_RECEIVE_HEADER:
         // Action
         // Receive Header data
         // 
         #receive(EN_R := (#ownInstance = #Config.instanceLock),
                  ID := #connection.ID,
                  LEN := #EIP_HEADER_LENGTH,
                  DATA := #receiveBuffer.Header);


         // Transition
         // Header received --> STATE_RECEIVE_DATA
         // Invalid Data --> IDLE
         // Error --> INIT
           IF #receive.NDR OR #receive.STATUS = #RESULT_SUCCESS THEN
             IF #receiveBuffer.Header.Length = 0 THEN
               //Unlocking MuteEx
               #Config.instanceLock := 0;
               #internalState := #STATE_IDLE;
             ELSE
               #internalState := #STATE_RECEIVE_DATA;
             END_IF;

           ELSIF #receive.STATUS <> #RESULT_IDLE AND
             #receive.STATUS <> #RESULT_JOB_RUNNING AND
             #receive.STATUS <> #RESULT_JOB_START AND
             #receive.STATUS <> #RESULT_SUCCESS
           THEN
             #Status := W#16#8300 OR (#receive.STATUS AND 16#00FF);
             #internalState := #STATE_IDLE;
           ELSE
             //Nothing to do, just wait here
             ;
           END_IF;

       #STATE_RECEIVE_DATA:
         // Action
         // Receive Data
         // 
         // assume job is still running
         #Status := #RESULT_JOB_RUNNING;

         #receive(EN_R := (#ownInstance = #Config.instanceLock),
                  ID := #connection.ID,
                  LEN := DWORD_TO_UINT(WORD_TO_DWORD(SWAP(UINT_TO_WORD(#receiveBuffer.Header.Length)))),
                  DATA := #receiveBuffer.Data);

         // Transition
         // Header received --> STATE_RECEIVE_DATA
         // Invalid Data --> IDLE
         // Error --> INIT

         IF #receive.NDR OR #receive.STATUS = #RESULT_SUCCESS THEN
           // Decode Response
           // 
           #currentResponse := SWAP(#receiveBuffer.Header.Command);

           //the Context will be a combination out of the own instance identifier
           //and a sequence number
           #receivedInstance := DWORD_TO_DINT(SHL(IN := USINT_TO_DWORD(#receiveBuffer.Header.Context[4]), N := 24) OR
                                              SHL(IN := USINT_TO_DWORD(#receiveBuffer.Header.Context[3]), N := 16) OR
                                              SHL(IN := USINT_TO_DWORD(#receiveBuffer.Header.Context[2]), N := 8) OR
                                              USINT_TO_DWORD(#receiveBuffer.Header.Context[1]));

           #receivedSequence := DWORD_TO_DINT(SHL(IN := USINT_TO_DWORD(#receiveBuffer.Header.Context[8]), N := 24) OR
                                              SHL(IN := USINT_TO_DWORD(#receiveBuffer.Header.Context[7]), N := 16) OR
                                              SHL(IN := USINT_TO_DWORD(#receiveBuffer.Header.Context[6]), N := 8) OR
                                              USINT_TO_DWORD(#receiveBuffer.Header.Context[5]));

           IF #currentResponse = #EIP_CMD_REG_SESSION THEN
             //Response to RegisterSession received
             // retrieve the SessionID (SessionHandle)
             IF #receiveBuffer.Header.Status = #EIP_STATUS_OK THEN
               #Config.currentSessionID := DWORD_TO_UDINT(SWAP(UDINT_TO_DWORD(#receiveBuffer.Header.SessionHandle)));
               #Status := #RESULT_SUCCESS;

             ELSE
               // inform the user about it
               // 
               #Status := W#16#7100 OR DWORD_TO_WORD((SHR(IN := UDINT_TO_DWORD(#receiveBuffer.Header.Status), N := 24)));

               //Cleaning up internal information and
               //gracefully disconnect
               IF #Config.currentSessionID = 0 THEN
                 // a previous session hasn't been established --> only disconnecting
                 #internalState := #STATE_DISCONNECTING;
               ELSE
                 // previous session existed (somehow) --> unregister before disconnecting
                 #internalState := #STATE_UNREGISTER_SESSION;
               END_IF;
             END_IF;

           ELSIF #currentResponse = #EIP_CMD_SEND_RR THEN
             //Response to Send RR Data received
             // determine Status of transmission
             // retrieve TagValue and DataType
             IF #receiveBuffer.Header.Status = #EIP_STATUS_OK THEN
               #itemLength := WORD_TO_INT(SHL(IN := USINT_TO_WORD(#receiveBuffer.Data[16]), N := 8) OR USINT_TO_WORD(#receiveBuffer.Data[15]));
               #currentCIPService := USINT_TO_BYTE(#receiveBuffer.Data[17]);
               IF #currentCIPService = (#CIP_SRV_TABLEREAD OR 16#80) AND
                 #receivedInstance = #ownInstance AND
                 #receivedSequence = #ownSequence
               THEN
                 //Check the status of the variable request
                 //  it may have failed on us (<>0)
                 //  
                 IF #receiveBuffer.Data[19] = #CIP_GENSTS_SUCCESS THEN

                   #receivedType := SHL(IN := USINT_TO_WORD(#receiveBuffer.Data[22]), N := 8) OR
                   USINT_TO_WORD(#receiveBuffer.Data[21]);

                   #valueIndex := 0;

                   WHILE #valueIndex <= (#itemLength - 6) DO

                     CASE WORD_TO_UINT(#receivedType) OF
                       #DT_BOOLEAN_ATOMIC:
                         // since it seems that there are difficulties accessing Booleans
                         // these accesses are being mapped into accesses to bytes (SINT)
                         // Therefore the code sections doubles here

                         #receivedValue.Short := USINT_TO_SINT(#receiveBuffer.Data[23 + #valueIndex]);

                         // only usable with S7-1500 or S7-1200 V4.x
                         //
                         #result := MOVE_BLK_VARIANT(SRC := #receivedValue.Short,
                                                     SRC_INDEX := 0,
                                                     DEST => #Value,
                                                     DEST_INDEX := #valueIndex,
                                                     COUNT := 1);
                         #valueIndex := #valueIndex + 1;
                         #DT_SINT_ATOMIC:
                         #receivedValue.Short := USINT_TO_SINT(#receiveBuffer.Data[23 + #valueIndex]);

                         // only usable with S7-1500 or S7-1200 V4.x
                         //
                         #result := MOVE_BLK_VARIANT(SRC := #receivedValue.Short,
                                                     SRC_INDEX := 0,
                                                     DEST => #Value,
                                                     DEST_INDEX := #valueIndex,
                                                     COUNT := 1);
                         #valueIndex := #valueIndex + 1;
                       #DT_INT_ATOMIC:
                         #receivedValue.Integer := WORD_TO_INT(SHL(IN := USINT_TO_WORD(#receiveBuffer.Data[24 + #valueIndex]), N := 8) OR
                                                                USINT_TO_WORD(#receiveBuffer.Data[23 + #valueIndex]));
                         // only usable with S7-1500 or S7-1200 V4.x
                         //          
                         #result := MOVE_BLK_VARIANT(SRC := #receivedValue.Integer,
                                                     SRC_INDEX := 0,
                                                     DEST => #Value,
                                                     DEST_INDEX := #valueIndex / 2,
                                                     COUNT := 1);
                         #valueIndex := #valueIndex + 2;
                       #DT_DINT_ATOMIC:
                         #receivedValue.Double := DWORD_TO_DINT(SHL(IN := USINT_TO_DWORD(#receiveBuffer.Data[26 + #valueIndex]), N := 24) OR
                                                                 SHL(IN := USINT_TO_DWORD(#receiveBuffer.Data[25 + #valueIndex]), N := 16) OR
                                                                 SHL(IN := USINT_TO_DWORD(#receiveBuffer.Data[24 + #valueIndex]), N := 8) OR
                                                                 USINT_TO_DWORD(#receiveBuffer.Data[23 + #valueIndex]));
                         // only usable with S7-1500 or S7-1200 V4.x
                         //          
                         #result := MOVE_BLK_VARIANT(SRC := #receivedValue.Double,
                                                     SRC_INDEX := 0,
                                                     DEST => #Value,
                                                     DEST_INDEX := #valueIndex / 4,
                                                     COUNT := 1);
                         #valueIndex := #valueIndex + 4;

                       #DT_FLOAT_ATOMIC:
                         #receivedValue.Float := DWORD_TO_REAL(SHL(IN := USINT_TO_DWORD(#receiveBuffer.Data[26 + #valueIndex]), N := 24) OR
                                                               SHL(IN := USINT_TO_DWORD(#receiveBuffer.Data[25 + #valueIndex]), N := 16) OR
                                                               SHL(IN := USINT_TO_DWORD(#receiveBuffer.Data[24 + #valueIndex]), N := 8) OR
                                                               USINT_TO_DWORD(#receiveBuffer.Data[23 + #valueIndex]));
                         // only usable with S7-1500 or S7-1200 V4.x
                         //          
                         #result := MOVE_BLK_VARIANT(SRC := #receivedValue.Float,
                                                     SRC_INDEX := 0,
                                                     DEST => #Value,
                                                     DEST_INDEX := #valueIndex / 4,
                                                     COUNT := 1);
                         #valueIndex := #valueIndex + 4;
                       ELSE
                         // throw warning
                         #Status := 0; //Unknown data type
                     END_CASE;


                   END_WHILE;

                   // show successful result
                   //
                   #Status := #RESULT_SUCCESS;

                   #NewData := TRUE;
                   IF #ownSequence = -1 THEN
                     #ownSequence := #ownSequence + 2;
                   ELSE
                     #ownSequence := #ownSequence + 1;
                   END_IF;

                 ELSIF #receiveBuffer.Data[19] = #CIP_GENSTS_PATH_DEST_UNKNOWN OR
                       #receiveBuffer.Data[19] = #CIP_GENSTS_PATH_SEG_ERROR
                 THEN
                   // throw warning
                   #Status := W#16#7200 OR USINT_TO_BYTE(#receiveBuffer.Data[19]);

                 ELSIF #receiveBuffer.Data[19] = #CIP_GENSTS_GENERIC THEN
                   #Status := W#16#7300 OR USINT_TO_BYTE(#receiveBuffer.Data[22]);
                 ELSE
                   // throw warning
                   #Status := W#16#72FF;  //Unknown error code
                 END_IF;

               ELSIF #currentCIPService = (#CIP_SRV_TABLEREAD_FRAG OR 16#80) THEN
                 #Status := W#16#7300 OR USINT_TO_BYTE(#receiveBuffer.Data[19]);

               ELSE
                 // throw warning
                 //   unexpected answer from host - ignoring it
                 #Status := W#16#8A00 OR #currentCIPService;
               END_IF;

             ELSE
               // inform the user about it
               // 
               #Status := W#16#7100 OR DWORD_TO_WORD((SHR(IN := UDINT_TO_DWORD(#receiveBuffer.Header.Status), N := 24)));

               //Cleaning up internal information and
               //gracefully disconnect
               IF #Config.currentSessionID = 0 THEN
                 // a previous session hasn't been established --> only disconnecting
                 #internalState := #STATE_DISCONNECTING;
               ELSE
                 // previous session existed (somehow) --> unregister before disconnecting
                 #internalState := #STATE_UNREGISTER_SESSION;
               END_IF;
             END_IF;
           ELSE
             //Unknown/ Unhandled Response received
             //  ignoring it
             #Status := W#16#8B00 OR #currentResponse;

             //#Config.currentSessionID := 0;
             //#internalState := #STATE_DISCONNECTING;
           END_IF;

           #receiveBuffer.Header.Length := 0;

           //Unlocking MuteEx
           #Config.instanceLock := 0;

           #internalState := #STATE_IDLE;
         ELSIF #receive.STATUS <> #RESULT_IDLE AND
               #receive.STATUS <> #RESULT_JOB_RUNNING AND
               #receive.STATUS <> #RESULT_JOB_START AND
               #receive.STATUS <> #RESULT_SUCCESS
         THEN
           #Status := W#16#8300 OR (#receive.STATUS AND 16#00FF);
           #internalState := #STATE_IDLE;
         ELSE
           //Nothing to do, just wait here
           ;
         END_IF;

       #STATE_UNREGISTER_SESSION:
         IF #Config.references = 1 THEN

           #sendBuffer.Header.Command := SWAP(#EIP_CMD_UNREG_SESSION);   //Command is RegisterSession (16#66)
           #sendBuffer.Header.Length := WORD_TO_UINT(SWAP(IN := UDINT_TO_WORD(#send.LEN - #EIP_HEADER_LENGTH)));    //Length of Data is 4 Bytes
           #sendBuffer.Header.SessionHandle := DWORD_TO_UDINT(SWAP(UDINT_TO_DWORD(#Config.currentSessionID)));
           #sendBuffer.Header.Status := 0;
           #sendBuffer.Header.Options := 0;
           //the Context will be a combination out of the own instance identifier
           //and a sequence number
           #sendBuffer.Header.Context[1] := DWORD_TO_USINT(DINT_TO_DWORD(#ownInstance) AND DW#16#000000FF);
           #sendBuffer.Header.Context[2] := DWORD_TO_USINT(SHR(IN := DINT_TO_DWORD(#ownInstance), N := 8) AND DW#16#000000FF);
           #sendBuffer.Header.Context[3] := DWORD_TO_USINT(SHR(IN := DINT_TO_DWORD(#ownInstance), N := 16) AND DW#16#000000FF);
           #sendBuffer.Header.Context[4] := DWORD_TO_USINT(SHR(IN := DINT_TO_DWORD(#ownInstance), N := 24) AND DW#16#000000FF);
           #sendBuffer.Header.Context[5] := DWORD_TO_USINT(DINT_TO_DWORD(#ownSequence) AND DW#16#000000FF);
           #sendBuffer.Header.Context[6] := DWORD_TO_USINT(SHR(IN := DINT_TO_DWORD(#ownSequence), N := 8) AND DW#16#000000FF);
           #sendBuffer.Header.Context[7] := DWORD_TO_USINT(SHR(IN := DINT_TO_DWORD(#ownSequence), N := 16) AND DW#16#000000FF);
           #sendBuffer.Header.Context[8] := DWORD_TO_USINT(SHR(IN := DINT_TO_DWORD(#ownSequence), N := 24) AND DW#16#000000FF);
           #sendBuffer.Data[1] := 16#00;

           //Checking the MuteEx
           IF #Config.instanceLock = 0 OR
             #Config.instanceLock = #ownInstance
           THEN
             //Locking the MutEx
             #Config.instanceLock := #ownInstance;
             #send.LEN := #EIP_HEADER_LENGTH;
             #send.REQ := TRUE;
             // Action
             // 

             #send(ID := #connection.ID,
                   DATA := #sendBuffer);

             // Transition
             //
             #internalState := #STATE_UNREGISTERING;
             #Config.references := #Config.references - 1;
           ELSE
             IF #Config.instanceLock = #ownInstance THEN
               #Config.instanceLock := 0;
             END_IF;
           END_IF;

         ELSE
           IF #Config.references > 1 THEN
             #Config.references := #Config.references - 1;
           END_IF;
           #internalState := #STATE_POWER_OFF;
         END_IF;

       #STATE_UNREGISTERING:
         // Action
         // 

         #send(ID := #connection.ID,
               DATA := #sendBuffer);

         // Transition
         //
         IF #send.STATUS = #RESULT_JOB_START THEN
           ;
         ELSIF #send.STATUS = #RESULT_JOB_RUNNING THEN
           #send.REQ := FALSE;

         ELSIF #send.STATUS = #RESULT_SUCCESS THEN
           #send.REQ := FALSE;
           #internalState := #STATE_DISCONNECTING;
           //Unlocking MuteEx
           #Config.instanceLock := 0;
         ELSE

           #Status := W#16#8200 OR (#send.STATUS AND 16#00FF);
           #send.REQ := FALSE;
           #internalState := #STATE_DISCONNECTING;
         END_IF;

